// TIA Portal project "TCC" (V14)

(* hardware
DEVICE "S71500/ET200MP station_1"  S7-1500 station
   slot 0: "Rail_0"  Rack  6ES7 590-1***0-0AA0
   slot 1: "Selection"  CPU 1516-3 PN/DP  6ES7 516-3AN01-0AB0  V2.1
      slot 3: "CPU display_1"  6ES7591-1BA00-0AA0
   slot 2: "DI 32x24VDC HF_1"  DI 32x24VDC HF  6ES7 521-1BL00-0AB0  V2.1
   slot 3: "DQ 32x24VDC/0.5A HF_1"  DQ 32x24VDC/0.5A HF  6ES7 522-1BL01-0AB0  V1.0
   slot 4: "AI 8xU/I/RTD/TC ST_1"  AI 8xU/I/RTD/TC ST  6ES7 531-7KF00-0AB0  V2.1
   slot 5: "AQ 4xU/I ST_1"  AQ 4xU/I ST  6ES7 532-5HD00-0AB0  V2.1
DEVICE "S71500/ET200MP station_2"  S7-1500 station
   slot 0: "Rail_0"  Rack  6ES7 590-1***0-0AA0
   slot 1: "Handling-Assembly-Storage"  CPU 1516-3 PN/DP  6ES7 516-3AN01-0AB0  V2.1
      slot 3: "CPU display_1"  6ES7591-1BA00-0AA0
   slot 2: "DI 32x24VDC HF_1"  DI 32x24VDC HF  6ES7 521-1BL00-0AB0  V2.1
   slot 3: "DQ 32x24VDC/0.5A HF_1"  DQ 32x24VDC/0.5A HF  6ES7 522-1BL01-0AB0  V1.0
   slot 4: "AI 8xU/I/RTD/TC ST_1"  AI 8xU/I/RTD/TC ST  6ES7 531-7KF00-0AB0  V2.1
   slot 5: "AQ 4xU/I ST_1"  AQ 4xU/I ST  6ES7 532-5HD00-0AB0  V2.1
   slot 6: "TM Count 2x24V_1"  TM Count 2x24V  6ES7 550-1AA00-0AB0  V1.1
*)

// ===== PLC "Selection"  CPU 1516-3 PN/DP =====

VAR_GLOBAL   // PLC tag table "Default tag table"
   "Clock_Byte" AT %MB25 : Byte;
   "Clock_10Hz" AT %M25.0 : Bool;
   "Clock_5Hz" AT %M25.1 : Bool;
   "Clock_2.5Hz" AT %M25.2 : Bool;
   "Clock_2Hz" AT %M25.3 : Bool;
   "Clock_1.25Hz" AT %M25.4 : Bool;
   "Clock_1Hz" AT %M25.5 : Bool;
   "Clock_0.625Hz" AT %M25.6 : Bool;
   "Clock_0.5Hz" AT %M25.7 : Bool;
END_VAR

VAR_GLOBAL   // PLC tag table "IOTAGS"
   "I_MAG1EXT" AT %I0.0 : Bool;   // MAG 1 Cylinder Extended
   "I_MAG1RET" AT %I0.1 : Bool;   // MAG 1 Cylinder Retracted
   "I_MAG1EMPT" AT %I0.2 : Bool;   // MAG 1 Empty
   "I_MAG2EXT" AT %I0.3 : Bool;   // MAG 2 Cylinder Extended
   "I_MAG2RET" AT %I0.4 : Bool;   // MAG 2 Cylinder Retracted
   "I_MAG2EMPT" AT %I0.5 : Bool;   // MAG 2 Empty
   "I_PSLD" AT %I2.0 : Bool;   // Proximity Sensor Left Discharge Cylinder
   "I_PSCD" AT %I2.1 : Bool;   // Proximity Sensor Center Discharge Cylinder
   "I_PSRD" AT %I2.2 : Bool;   // Proximity Sensor Right Discharge Cylinder
   "I_RELAY1" AT %I2.3 : Bool;   // Relay
   "I_LDCEXT" AT %I1.0 : Bool;   // Left Discharge Cylinder Extended
   "I_LDCRET" AT %I1.1 : Bool;   // Left Discharge Cylinder Retracted
   "I_CDCEXT" AT %I1.2 : Bool;   // Center Discharge Cylinder Extended
   "I_CDCRET" AT %I1.3 : Bool;   // Center Discharge Cylinder Retracted
   "I_RDCEXT" AT %I1.4 : Bool;   // Right Discharge Cylinder Extended
   "I_RDCRET" AT %I1.5 : Bool;   // Right Discharge Cylinder Retracted
   "I_WHIT" AT %I1.6 : Bool;   // White Color Sensor
   "I_METAL" AT %I1.7 : Bool;   // Metalic Sensor
   "I_PSEOC" AT %I0.6 : Bool;   // Proximity Sensor End Of Conveyor Belt
   "I_DS" AT %IW4 : Word;   // Distance Sensor
   "O_MAG1EXT" AT %Q1.0 : Bool;   // Extend MAG 1 Cylinder
   "O_MAG1RET" AT %Q1.1 : Bool;   // Retract MAG 1 Cylinder
   "O_MAG2EXT" AT %Q1.2 : Bool;   // Extend MAG 2 Cylinder
   "O_MAG2RET" AT %Q1.3 : Bool;   // Retra MAG 2 Cylinder
   "O_RDCEXT" AT %Q0.2 : Bool;   // Extend Right Discharge Cylinder
   "O_CDCEXT" AT %Q0.1 : Bool;   // Extend Center Discharge Cylinder
   "O_LDCEXT" AT %Q0.0 : Bool;   // Extend Left Discharge Cylinder
   "O_CBFW" AT %Q1.4 : Bool;   // Conveyor Belt Forward
   "O_CBREV" AT %Q1.5 : Bool;   // Conveyor Belt Reverse
END_VAR

VAR_GLOBAL   // PLC tag table "Places"
   "p0" AT %M0.0 : Bool;
   "p1" AT %M0.1 : Bool;
   "p2" AT %M0.2 : Bool;
   "p3" AT %M0.3 : Bool;
   "p4" AT %M0.4 : Bool;
   "p5" AT %M0.5 : Bool;
   "p6" AT %M0.6 : Bool;
   "p7" AT %M0.7 : Bool;
   "p8" AT %M1.0 : Bool;
   "p9" AT %M1.1 : Bool;
   "p10" AT %M1.2 : Bool;
   "p11" AT %M1.3 : Bool;
   "p12" AT %M1.4 : Bool;
   "p27" AT %M1.6 : Bool;
   "p28" AT %M1.7 : Bool;
   "p29" AT %M2.0 : Bool;
   "p30" AT %M2.1 : Bool;
   "p31" AT %M2.2 : Bool;
   "p32" AT %M2.3 : Bool;
   "p33" AT %M2.4 : Bool;
   "p34" AT %M2.5 : Bool;
   "p35" AT %M2.6 : Bool;
   "p36" AT %M2.7 : Bool;
   "p37" AT %M3.0 : Bool;
   "p38" AT %M3.1 : Bool;
   "p39" AT %M3.2 : Bool;
   "p40" AT %M3.3 : Bool;
   "p41" AT %M3.4 : Bool;
   "p42" AT %M3.5 : Bool;
   "p43" AT %M3.6 : Bool;
   "p44" AT %M3.7 : Bool;
   "p45" AT %M4.0 : Bool;
   "p46" AT %M4.1 : Bool;
   "p47" AT %M4.2 : Bool;
   "p48" AT %M4.3 : Bool;
   "p49" AT %M4.4 : Bool;
   "p50" AT %M4.5 : Bool;
   "p51" AT %M4.6 : Bool;
   "p52" AT %M4.7 : Bool;
   "p53" AT %M5.0 : Bool;
   "p54" AT %M5.1 : Bool;
   "p55" AT %M5.2 : Bool;
   "p56" AT %M5.3 : Bool;
   "p57" AT %M5.4 : Bool;
   "p58" AT %M5.5 : Bool;
   "p59" AT %M5.6 : Bool;
   "p60" AT %M5.7 : Bool;
   "p61" AT %M6.0 : Bool;
   "p62" AT %M6.1 : Bool;
   "p63" AT %M6.2 : Bool;
   "p64" AT %M6.3 : Bool;
   "p65" AT %M6.4 : Bool;
   "p66" AT %M6.5 : Bool;
   "p67" AT %M6.6 : Bool;
   "p68" AT %M6.7 : Bool;
   "p69" AT %M7.0 : Bool;
   "p70" AT %M7.1 : Bool;
   "p71" AT %M7.2 : Bool;
   "p72" AT %M7.3 : Bool;
   "p73" AT %M7.4 : Bool;
END_VAR

VAR_GLOBAL   // PLC tag table "Transitions"
   "t0" AT %M7.5 : Bool;
   "t1" AT %M7.6 : Bool;
   "t2" AT %M7.7 : Bool;
   "t3" AT %M8.0 : Bool;
   "t4" AT %M8.1 : Bool;
   "t5" AT %M8.2 : Bool;
   "t6" AT %M8.3 : Bool;
   "t7" AT %M8.4 : Bool;
   "t18" AT %M8.5 : Bool;
   "t19" AT %M8.6 : Bool;
   "t20" AT %M8.7 : Bool;
   "t21" AT %M9.0 : Bool;
   "t22" AT %M9.1 : Bool;
   "t23" AT %M9.2 : Bool;
   "t24" AT %M9.3 : Bool;
   "t25" AT %M9.4 : Bool;
   "t26" AT %M9.5 : Bool;
   "t27" AT %M9.6 : Bool;
   "t28" AT %M9.7 : Bool;
   "t29" AT %M10.0 : Bool;
   "t30" AT %M10.1 : Bool;
   "t31" AT %M10.2 : Bool;
   "t32" AT %M10.3 : Bool;
   "t33" AT %M10.4 : Bool;
   "t34" AT %M10.5 : Bool;
   "t35" AT %M10.6 : Bool;
   "t36" AT %M10.7 : Bool;
   "t37" AT %M11.0 : Bool;
   "t38" AT %M11.1 : Bool;
   "t39" AT %M11.2 : Bool;
   "t40" AT %M11.3 : Bool;
   "t41" AT %M11.4 : Bool;
   "t42" AT %M11.5 : Bool;
   "t43" AT %M11.6 : Bool;
   "t44" AT %M11.7 : Bool;
   "t45" AT %M12.0 : Bool;
   "t46" AT %M12.1 : Bool;
   "t47" AT %M12.2 : Bool;
   "t48" AT %M12.3 : Bool;
   "t49" AT %M12.4 : Bool;
   "t50" AT %M12.5 : Bool;
   "t51" AT %M12.6 : Bool;
   "t52" AT %M12.7 : Bool;
   "t53" AT %M13.0 : Bool;
   "t54" AT %M13.1 : Bool;
   "t55" AT %M13.2 : Bool;
   "t56" AT %M13.3 : Bool;
   "t57" AT %M13.4 : Bool;
   "t58" AT %M13.5 : Bool;
   "t59" AT %M13.6 : Bool;
   "t60" AT %M13.7 : Bool;
   "t61" AT %M14.0 : Bool;
   "t62" AT %M14.1 : Bool;
   "t63" AT %M14.2 : Bool;
   "t64" AT %M14.3 : Bool;
   "t65" AT %M14.4 : Bool;
   "t66" AT %M14.5 : Bool;
   "t67" AT %M14.6 : Bool;
   "t68" AT %M14.7 : Bool;
   "t69" AT %M15.0 : Bool;
   "t70" AT %M15.1 : Bool;
   "t71" AT %M15.2 : Bool;
END_VAR

VAR_GLOBAL   // PLC tag table "Auxiliar"
   "PresenceR" AT %M15.3 : Bool;
   "ConcUP" AT %M15.4 : Bool;
   "ConcDWN" AT %M15.5 : Bool;
   "Presence_prev" AT %M15.6 : Bool;
   "I_PSEOCr_prev" AT %M15.7 : Bool;
   "PSEOCR" AT %M16.0 : Bool;
   "PSEOCF" AT %M16.1 : Bool;
   "BTInit" AT %M24.0 : Bool;
   "BTStart" AT %M24.1 : Bool;
   "BTSTOP" AT %M24.2 : Bool;
   "btget" AT %M24.3 : Bool;
   "bini" AT %M1.5 : Bool;
   "clkprev" AT %M24.4 : Bool;
   "I_PSEOCf_prev" AT %M24.6 : Bool;
END_VAR

VAR_GLOBAL   // PLC tag table "Conditions"
   "b0" AT %M16.2 : Bool;
   "b1" AT %M16.3 : Bool;
   "b2" AT %M16.4 : Bool;
   "b3" AT %M16.5 : Bool;
   "b4" AT %M16.6 : Bool;
   "b5" AT %M16.7 : Bool;
   "b6" AT %M17.0 : Bool;
   "b7" AT %M17.1 : Bool;
   "b18" AT %M17.2 : Bool;
   "b19" AT %M17.3 : Bool;
   "b20" AT %M17.4 : Bool;
   "b21" AT %M17.5 : Bool;
   "b22" AT %M17.6 : Bool;
   "b23" AT %M17.7 : Bool;
   "b24" AT %M18.0 : Bool;
   "b25" AT %M18.1 : Bool;
   "b26" AT %M18.2 : Bool;
   "b27" AT %M18.3 : Bool;
   "b28" AT %M18.4 : Bool;
   "b29" AT %M18.5 : Bool;
   "b30" AT %M18.6 : Bool;
   "b31" AT %M18.7 : Bool;
   "b32" AT %M19.0 : Bool;
   "b33" AT %M19.1 : Bool;
   "b34" AT %M19.2 : Bool;
   "b35" AT %M19.3 : Bool;
   "b36" AT %M19.4 : Bool;
   "b37" AT %M19.5 : Bool;
   "b38" AT %M19.6 : Bool;
   "b39" AT %M19.7 : Bool;
   "b40" AT %M20.0 : Bool;
   "b41" AT %M20.1 : Bool;
   "b42" AT %M20.2 : Bool;
   "b43" AT %M20.3 : Bool;
   "b44" AT %M20.4 : Bool;
   "b45" AT %M20.5 : Bool;
   "b46" AT %M20.6 : Bool;
   "b47" AT %M20.7 : Bool;
   "b48" AT %M21.0 : Bool;
   "b49" AT %M21.1 : Bool;
   "b50" AT %M21.2 : Bool;
   "b51" AT %M21.3 : Bool;
   "b52" AT %M21.4 : Bool;
   "b53" AT %M21.5 : Bool;
   "b54" AT %M21.6 : Bool;
   "b55" AT %M21.7 : Bool;
   "b56" AT %M22.0 : Bool;
   "b57" AT %M22.1 : Bool;
   "b58" AT %M22.2 : Bool;
   "b59" AT %M22.3 : Bool;
   "b60" AT %M22.4 : Bool;
   "b61" AT %M22.5 : Bool;
   "b62" AT %M22.6 : Bool;
   "b63" AT %M22.7 : Bool;
   "b64" AT %M23.0 : Bool;
   "b65" AT %M23.1 : Bool;
   "b66" AT %M23.2 : Bool;
   "b67" AT %M23.3 : Bool;
   "b68" AT %M23.4 : Bool;
   "b69" AT %M23.5 : Bool;
   "b70" AT %M23.6 : Bool;
   "b71" AT %M23.7 : Bool;
   "b162" AT %M24.5 : Bool;
   "b156_StopAll" AT %M24.7 : Bool;
END_VAR

VAR_GLOBAL   // PLC tag table "Logging"
   "AcqRun" AT %M26.0 : Bool;
   "stopAcquisition" AT %M26.2 : Bool;
   "DataLogCreated" AT %M26.3 : Bool;
   "Done_Signal" AT %M26.4 : Bool;
   "Busy" AT %M26.5 : Bool;
   "Error" AT %M26.6 : Bool;
   "Status" AT %MW28 : Word;
   "LogTimeElapsed" AT %MD30 : Time;
   "AcqNewValues" AT %M26.7 : Bool;
   "Done_Open" AT %M27.0 : Bool;
   "Busy_Open" AT %M27.1 : Bool;
   "Error_Open" AT %M27.2 : Bool;
   "Status_Open" AT %MW34 : Word;
   "Done_Write" AT %M36.0 : Bool;
   "Busy_Write" AT %M36.1 : Bool;
   "Error_Write" AT %M36.2 : Bool;
   "Status_Write" AT %MW38 : Word;
   "closeDL" AT %M27.3 : Bool;
   "startAcquisition" AT %M26.1 : Bool;
   "DeleteDl" AT %M27.4 : Bool;
   "startAcqprev" AT %M27.5 : Bool;
END_VAR

// folder: Logging

DATA_BLOCK "LOGDATA_DB"   // DB18
{ S7_Optimized_Access := 'TRUE' }
VERSION : 0.1
// stored: InstanceOfName LOGDATA
"LOGDATA"
BEGIN
END_DATA_BLOCK

DATA_BLOCK "IOVEC_FROMPLC2"   // DB19
{ S7_Optimized_Access := 'FALSE' }
VERSION : 0.1
   VAR
      I_SDO : Bool;
      I_SDC : Bool;
      I_AUHEXT : Bool;
      I_AUHRET : Bool;
      I_INDARM : Bool;
      I_ARMLOW : Bool;
      I_ARMHIG : Bool;
      I_ARMRET : Bool;
      I_ARMEXT : Bool;
      I_SUVE : Bool;
      I_SUILS : Bool;
      I_SUSLS : Bool;
      I_SUEXT : Bool;
      I_SURET : Bool;
      I_RELAY2 : Bool;
      I_SUHE : Bool;
      I_SURLS : Bool;
      I_SULLS : Bool;
      I_SUARMALE : Bool;
      O_SDO : Bool;
      O_SDC : Bool;
      O_AUHRET : Bool;
      O_AUHEXT : Bool;
      O_PRESSLOW : Bool;
      O_PRESSHIG : Bool;
      O_ARMHIG : Bool;
      O_VACON : Bool;
      O_ARMEXT : Bool;
      O_ARMCCW : Bool;
      O_ARMCW : Bool;
      O_SUEXT : Bool;
      O_SUUP : Bool;
      O_SUDWN : Bool;
      O_SURIGHT : Bool;
      O_SULEFT : Bool;
   END_VAR
BEGIN
END_DATA_BLOCK

DATA_BLOCK "DATALOGDATA"   // DB21
{ S7_Optimized_Access := 'TRUE' }
VERSION : 0.1
   VAR
      IOVECNAMES : Array[0..64] of String;
      IOVEC : Array[0..64] of Bool;
      AcqValues : Array[0..64] of Bool;
      AcqValuesprev : Array[0..64] of Bool;
      Data : Struct
         I_MAG1EXT : Bool;
         I_MAG1RET : Bool;
         I_MAG1EMPT : Bool;
         I_MAG2EXT : Bool;
         I_MAG2RET : Bool;
         I_MAG2EMPT : Bool;
         I_PSLD : Bool;
         I_PSCD : Bool;
         I_PSRD : Bool;
         I_RELAY1 : Bool;
         I_LDCEXT : Bool;
         I_LDCRET : Bool;
         I_CDCEXT : Bool;
         I_CDCRET : Bool;
         I_RDCEXT : Bool;
         I_RDCRET : Bool;
         I_WHIT : Bool;
         I_METAL : Bool;
         I_PSEOC : Bool;
         ConcDWN : Bool;
         ConcUP : Bool;
         O_MAG1EXT : Bool;
         O_MAG1RET : Bool;
         O_MAG2EXT : Bool;
         O_MAG2RET : Bool;
         O_RDCEXT : Bool;
         O_CDCEXT : Bool;
         O_LDCEXT : Bool;
         O_CBFW : Bool;
         O_CBREV : Bool;
         I_SDO : Bool;
         I_SDC : Bool;
         I_AUHEXT : Bool;
         I_AUHRET : Bool;
         I_INDARM : Bool;
         I_ARMLOW : Bool;
         I_ARMHIG : Bool;
         I_ARMRET : Bool;
         I_ARMEXT : Bool;
         I_SUVE : Bool;
         I_SUILS : Bool;
         I_SUSLS : Bool;
         I_SUEXT : Bool;
         I_SURET : Bool;
         I_RELAY2 : Bool;
         I_SUHE : Bool;
         I_SURLS : Bool;
         I_SULLS : Bool;
         I_SUARMALE : Bool;
         O_SDO : Bool;
         O_SDC : Bool;
         O_AUHRET : Bool;
         O_AUHEXT : Bool;
         O_PRESSLOW : Bool;
         O_PRESSHIG : Bool;
         O_ARMHIG : Bool;
         O_VACON : Bool;
         O_ARMEXT : Bool;
         O_ARMCCW : Bool;
         O_ARMCW : Bool;
         O_SUEXT : Bool;
         O_SUUP : Bool;
         O_SUDWN : Bool;
         O_SURIGHT : Bool;
         O_SULEFT : Bool;
      END_STRUCT;
      header : String;
      ID : DWord;
      "Name" : String;
   END_VAR
BEGIN
   IOVECNAMES[1] := '1';
   IOVECNAMES[2] := '2';
   IOVECNAMES[3] := '3';
   IOVECNAMES[4] := '4';
   IOVECNAMES[5] := '5';
   IOVECNAMES[6] := '6';
   IOVECNAMES[7] := '7';
   IOVECNAMES[8] := '8';
   IOVECNAMES[9] := '9';
   IOVECNAMES[10] := '10';
   IOVECNAMES[11] := '11';
   IOVECNAMES[12] := '12';
   IOVECNAMES[13] := '13';
   IOVECNAMES[14] := '14';
   IOVECNAMES[15] := '15';
   IOVECNAMES[16] := '16';
   IOVECNAMES[17] := '17';
   IOVECNAMES[18] := '18';
   IOVECNAMES[19] := '19';
   IOVECNAMES[20] := '20';
   IOVECNAMES[21] := '21';
   IOVECNAMES[22] := '22';
   IOVECNAMES[0] := '0';
   IOVECNAMES[23] := '23';
   IOVECNAMES[24] := '24';
   IOVECNAMES[25] := '25';
   IOVECNAMES[26] := '26';
   IOVECNAMES[27] := '27';
   IOVECNAMES[28] := '28';
   IOVECNAMES[29] := '29';
   IOVECNAMES[30] := '30';
   IOVECNAMES[31] := '31';
   IOVECNAMES[32] := '32';
   IOVECNAMES[33] := '33';
   IOVECNAMES[34] := '34';
   IOVECNAMES[35] := '35';
   IOVECNAMES[36] := '36';
   IOVECNAMES[37] := '37';
   IOVECNAMES[38] := '38';
   IOVECNAMES[39] := '39';
   IOVECNAMES[40] := '40';
   IOVECNAMES[41] := '41';
   IOVECNAMES[42] := '42';
   IOVECNAMES[43] := '43';
   IOVECNAMES[44] := '44';
   IOVECNAMES[45] := '45';
   IOVECNAMES[46] := '46';
   IOVECNAMES[47] := '47';
   IOVECNAMES[48] := '48';
   IOVECNAMES[49] := '49';
   IOVECNAMES[50] := '50';
   IOVECNAMES[51] := '51';
   IOVECNAMES[52] := '52';
   IOVECNAMES[53] := '53';
   IOVECNAMES[54] := '54';
   IOVECNAMES[55] := '55';
   IOVECNAMES[56] := '56';
   IOVECNAMES[57] := '57';
   IOVECNAMES[58] := '58';
   IOVECNAMES[59] := '59';
   IOVECNAMES[60] := '60';
   IOVECNAMES[61] := '61';
   IOVECNAMES[62] := '62';
   IOVECNAMES[63] := '63';
   IOVECNAMES[64] := '64';
END_DATA_BLOCK

// folder: PetriNet

DATA_BLOCK "FROM_PLC2"   // DB4
{ S7_Optimized_Access := 'FALSE' }
VERSION : 0.1
   VAR
      p13 : Bool;
      p17 : Bool;
      p26 : Bool;
      p14 : Bool;
      p18 : Bool;
      p107 : Bool;
      p0 : Bool;
      b162aux : Bool;
   END_VAR
BEGIN
END_DATA_BLOCK

DATA_BLOCK "TO_PLC2"   // DB5
{ S7_Optimized_Access := 'FALSE' }
VERSION : 0.1
   VAR
      b0 : Bool;
      b18 : Bool;
      b19 : Bool;
      b71 : Bool;
      b45 : Bool;
      b162 : Bool;
      btStopOn : Bool;
      btStopOff : Bool;
   END_VAR
BEGIN
END_DATA_BLOCK

// folder: PetriNet/TimedTransitions

DATA_BLOCK "t7_time"   // DB1
{ S7_Optimized_Access := 'TRUE' }
AUTHOR : Simatic
FAMILY : IEC
NAME : IEC_TMR
VERSION : 1.0
// stored: InstanceOfName IEC_TIMER
"IEC_TIMER"
BEGIN
END_DATA_BLOCK

DATA_BLOCK "t24_time"   // DB6
{ S7_Optimized_Access := 'TRUE' }
AUTHOR : Simatic
FAMILY : IEC
NAME : IEC_TMR
VERSION : 1.0
// stored: InstanceOfName IEC_TIMER
"IEC_TIMER"
BEGIN
END_DATA_BLOCK

DATA_BLOCK "t25_time"   // DB7
{ S7_Optimized_Access := 'TRUE' }
AUTHOR : Simatic
FAMILY : IEC
NAME : IEC_TMR
VERSION : 1.0
// stored: InstanceOfName IEC_TIMER
"IEC_TIMER"
BEGIN
END_DATA_BLOCK

DATA_BLOCK "t43_time"   // DB8
{ S7_Optimized_Access := 'TRUE' }
AUTHOR : Simatic
FAMILY : IEC
NAME : IEC_TMR
VERSION : 1.0
// stored: InstanceOfName IEC_TIMER
"IEC_TIMER"
BEGIN
END_DATA_BLOCK

DATA_BLOCK "t50_time"   // DB9
{ S7_Optimized_Access := 'TRUE' }
AUTHOR : Simatic
FAMILY : IEC
NAME : IEC_TMR
VERSION : 1.0
// stored: InstanceOfName IEC_TIMER
"IEC_TIMER"
BEGIN
END_DATA_BLOCK

DATA_BLOCK "t51_time"   // DB10
{ S7_Optimized_Access := 'TRUE' }
AUTHOR : Simatic
FAMILY : IEC
NAME : IEC_TMR
VERSION : 1.0
// stored: InstanceOfName IEC_TIMER
"IEC_TIMER"
BEGIN
END_DATA_BLOCK

DATA_BLOCK "t69_time"   // DB11
{ S7_Optimized_Access := 'TRUE' }
AUTHOR : Simatic
FAMILY : IEC
NAME : IEC_TMR
VERSION : 1.0
// stored: InstanceOfName IEC_TIMER
"IEC_TIMER"
BEGIN
END_DATA_BLOCK

// folder: System blocks/Program resources

DATA_BLOCK "LogTime"   // DB12
{ S7_Optimized_Access := 'TRUE' }
AUTHOR : Simatic
FAMILY : IEC
NAME : IEC_TMR
VERSION : 1.0
// stored: InstanceOfName IEC_TIMER
"IEC_TIMER"
BEGIN
END_DATA_BLOCK

// folder: (top level)

ORGANIZATION_BLOCK "Main"   // OB1, LAD, ProgramCycle
TITLE = "Main Program Sweep (Cycle)"
{ S7_Optimized_Access := 'TRUE' }
VERSION : 0.1
   VAR_INPUT
      Initial_Call : Bool;   // Initial call of this OB
      Remanence : Bool;   // =True, if remanent data are available
   END_VAR
BEGIN

REGION Network 1: GET VALUES FROM OTHER PLC
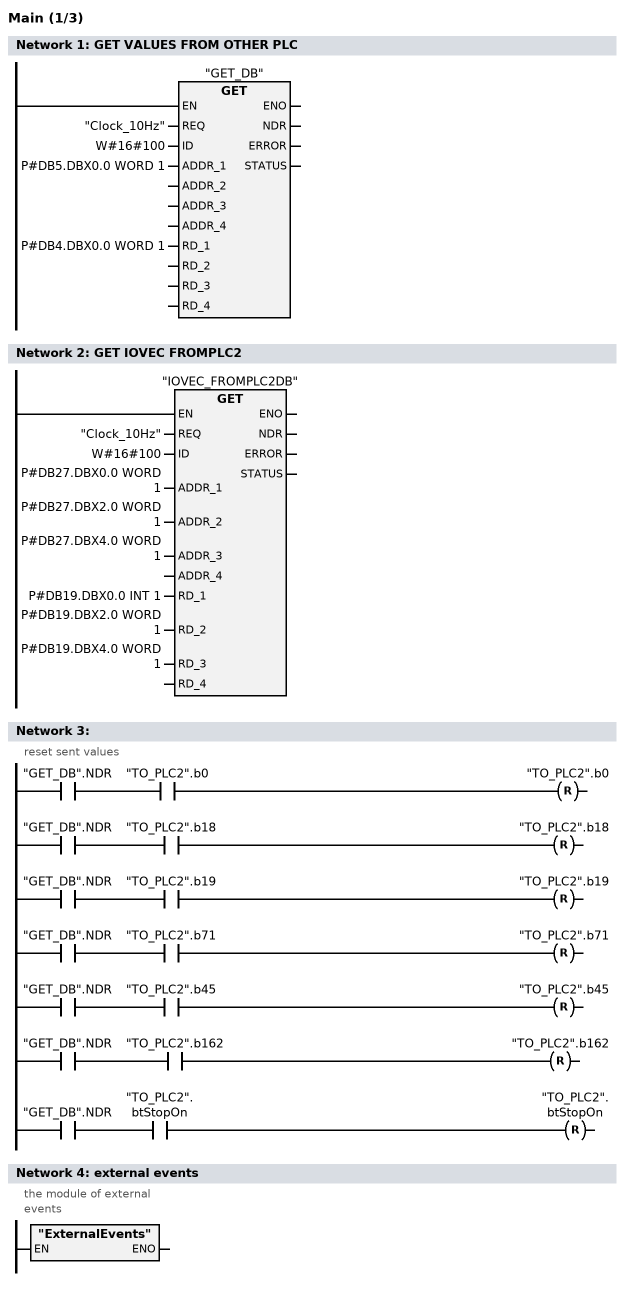
   "GET_DB"(REQ := "Clock_10Hz", ID := W#16#100, ADDR_1 := P#DB5.DBX0.0 WORD 1, RD_1 := P#DB4.DBX0.0 WORD 1);   // GET
END_REGION

REGION Network 2: GET IOVEC FROMPLC2
   "IOVEC_FROMPLC2DB"(REQ := "Clock_10Hz",   // GET
                      ID := W#16#100,
                      ADDR_1 := P#DB27.DBX0.0 WORD 1,
                      ADDR_2 := P#DB27.DBX2.0 WORD 1,
                      ADDR_3 := P#DB27.DBX4.0 WORD 1,
                      RD_1 := P#DB19.DBX0.0 INT 1,
                      RD_2 := P#DB19.DBX2.0 WORD 1,
                      RD_3 := P#DB19.DBX4.0 WORD 1);
END_REGION

REGION Network 3
   // reset sent values
   RUNG wire#powerrail
      Contact( "GET_DB".NDR )
      Contact( "TO_PLC2".b0 )
      R_Coil( "TO_PLC2".b0 )
   END_RUNG
   RUNG wire#powerrail
      Contact( "GET_DB".NDR )
      Contact( "TO_PLC2".b18 )
      R_Coil( "TO_PLC2".b18 )
   END_RUNG
   RUNG wire#powerrail
      Contact( "GET_DB".NDR )
      Contact( "TO_PLC2".b19 )
      R_Coil( "TO_PLC2".b19 )
   END_RUNG
   RUNG wire#powerrail
      Contact( "GET_DB".NDR )
      Contact( "TO_PLC2".b71 )
      R_Coil( "TO_PLC2".b71 )
   END_RUNG
   RUNG wire#powerrail
      Contact( "GET_DB".NDR )
      Contact( "TO_PLC2".b45 )
      R_Coil( "TO_PLC2".b45 )
   END_RUNG
   RUNG wire#powerrail
      Contact( "GET_DB".NDR )
      Contact( "TO_PLC2".b162 )
      R_Coil( "TO_PLC2".b162 )
   END_RUNG
   RUNG wire#powerrail
      Contact( "GET_DB".NDR )
      Contact( "TO_PLC2".btStopOn )
      R_Coil( "TO_PLC2".btStopOn )
   END_RUNG
   // the same network as SCL:
   IF "GET_DB".NDR AND "TO_PLC2".b0 THEN "TO_PLC2".b0 := FALSE; END_IF;
   IF "GET_DB".NDR AND "TO_PLC2".b18 THEN "TO_PLC2".b18 := FALSE; END_IF;
   IF "GET_DB".NDR AND "TO_PLC2".b19 THEN "TO_PLC2".b19 := FALSE; END_IF;
   IF "GET_DB".NDR AND "TO_PLC2".b71 THEN "TO_PLC2".b71 := FALSE; END_IF;
   IF "GET_DB".NDR AND "TO_PLC2".b45 THEN "TO_PLC2".b45 := FALSE; END_IF;
   IF "GET_DB".NDR AND "TO_PLC2".b162 THEN "TO_PLC2".b162 := FALSE; END_IF;
   IF "GET_DB".NDR AND "TO_PLC2".btStopOn THEN "TO_PLC2".btStopOn := FALSE; END_IF;
END_REGION

REGION Network 4: external events
   // the module of external
   // events
   RUNG wire#powerrail
      "ExternalEvents"()
   END_RUNG
   // the same network as SCL:
   "ExternalEvents"();
END_REGION

REGION Network 5: conditions
   // the module of firing conditions
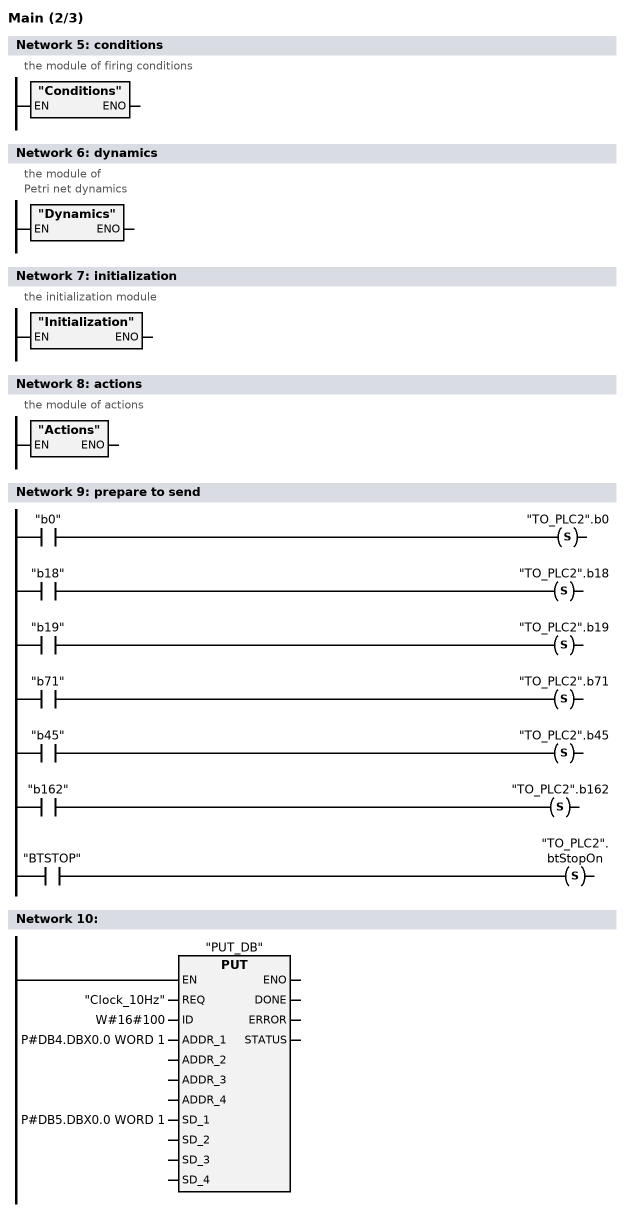
   RUNG wire#powerrail
      "Conditions"()
   END_RUNG
   // the same network as SCL:
   "Conditions"();
END_REGION

REGION Network 6: dynamics
   // the module of
   // Petri net dynamics
   RUNG wire#powerrail
      "Dynamics"()
   END_RUNG
   // the same network as SCL:
   "Dynamics"();
END_REGION

REGION Network 7: initialization
   // the initialization module
   RUNG wire#powerrail
      "Initialization"()
   END_RUNG
   // the same network as SCL:
   "Initialization"();
END_REGION

REGION Network 8: actions
   // the module of actions
   RUNG wire#powerrail
      "Actions"()
   END_RUNG
   // the same network as SCL:
   "Actions"();
END_REGION

REGION Network 9: prepare to send
   RUNG wire#powerrail
      Contact( "b0" )
      S_Coil( "TO_PLC2".b0 )
   END_RUNG
   RUNG wire#powerrail
      Contact( "b18" )
      S_Coil( "TO_PLC2".b18 )
   END_RUNG
   RUNG wire#powerrail
      Contact( "b19" )
      S_Coil( "TO_PLC2".b19 )
   END_RUNG
   RUNG wire#powerrail
      Contact( "b71" )
      S_Coil( "TO_PLC2".b71 )
   END_RUNG
   RUNG wire#powerrail
      Contact( "b45" )
      S_Coil( "TO_PLC2".b45 )
   END_RUNG
   RUNG wire#powerrail
      Contact( "b162" )
      S_Coil( "TO_PLC2".b162 )
   END_RUNG
   RUNG wire#powerrail
      Contact( "BTSTOP" )
      S_Coil( "TO_PLC2".btStopOn )
   END_RUNG
   // the same network as SCL:
   IF "b0" THEN "TO_PLC2".b0 := TRUE; END_IF;
   IF "b18" THEN "TO_PLC2".b18 := TRUE; END_IF;
   IF "b19" THEN "TO_PLC2".b19 := TRUE; END_IF;
   IF "b71" THEN "TO_PLC2".b71 := TRUE; END_IF;
   IF "b45" THEN "TO_PLC2".b45 := TRUE; END_IF;
   IF "b162" THEN "TO_PLC2".b162 := TRUE; END_IF;
   IF "BTSTOP" THEN "TO_PLC2".btStopOn := TRUE; END_IF;
END_REGION

REGION Network 10
   "PUT_DB"(REQ := "Clock_10Hz", ID := W#16#100, ADDR_1 := P#DB4.DBX0.0 WORD 1, SD_1 := P#DB5.DBX0.0 WORD 1);   // PUT
END_REGION

REGION Network 11: LOG DATA
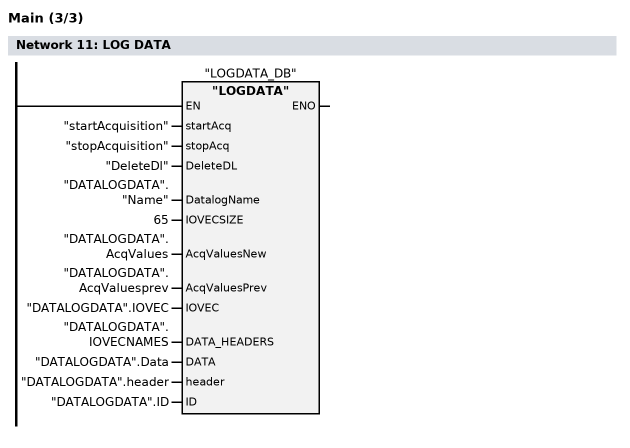
   RUNG wire#powerrail
      "LOGDATA_DB"(startAcq := "startAcquisition", stopAcq := "stopAcquisition", DeleteDL := "DeleteDl", DatalogName := "DATALOGDATA"."Name", IOVECSIZE := 65, AcqValuesNew := "DATALOGDATA".AcqValues, AcqValuesPrev := "DATALOGDATA".AcqValuesprev, IOVEC := "DATALOGDATA".IOVEC, DATA_HEADERS := "DATALOGDATA".IOVECNAMES, DATA := "DATALOGDATA".Data, header := "DATALOGDATA".header, ID := "DATALOGDATA".ID)
   END_RUNG
   // the same network as SCL:
   "LOGDATA_DB"(startAcq := "startAcquisition",   // "LOGDATA"
                stopAcq := "stopAcquisition",
                DeleteDL := "DeleteDl",
                DatalogName := "DATALOGDATA"."Name",
                IOVECSIZE := 65,
                AcqValuesNew := "DATALOGDATA".AcqValues,
                AcqValuesPrev := "DATALOGDATA".AcqValuesprev,
                IOVEC := "DATALOGDATA".IOVEC,
                DATA_HEADERS := "DATALOGDATA".IOVECNAMES,
                DATA := "DATALOGDATA".Data,
                header := "DATALOGDATA".header,
                ID := "DATALOGDATA".ID);
END_REGION
END_ORGANIZATION_BLOCK

// folder: Logging

FUNCTION_BLOCK "LOGDATA"   // FB1, LAD
{ S7_Optimized_Access := 'TRUE' }
VERSION : 0.1
   VAR_INPUT
      startAcq : Bool;
      stopAcq : Bool;
      DeleteDL : Bool;
      DatalogName : String;
      IOVECSIZE : UDInt;
   END_VAR
   VAR_IN_OUT
      AcqValuesNew : Array[*] of Bool;
      AcqValuesPrev : Array[*] of Bool;
      IOVEC : Array[*] of Bool;
      DATA_HEADERS : Array[*] of String;
      DATA : Variant;
      header : String;
      ID : DWord;
   END_VAR
   VAR_TEMP
      DeleteDatalog : Bool;
      moveBlkVariantRetVal : Int;
      i : Int;
      dataheaderslowerbound : DInt;
      dataheadersupperbound : DInt;
   END_VAR
   VAR_TEMP   // added for the SCL form of the ladder/FBD networks
      _w1 : Bool;
      _w2 : Bool;
   END_VAR
BEGIN

REGION Network 1 (SCL): Name header
       #header := '';
   #dataheaderslowerbound := LOWER_BOUND(ARR := #DATA_HEADERS, DIM := 1);
   #dataheadersupperbound := UPPER_BOUND(ARR := #DATA_HEADERS, DIM := 1);

   FOR #i := #dataheaderslowerbound TO #dataheadersupperbound-1 DO
       // Statement section FOR

       #header := CONCAT(IN1 := #header, IN2 := #DATA_HEADERS[#i]);
       #header := CONCAT(IN1 := #header, IN2 := ',');
   END_FOR;
   #header := CONCAT(IN1 := #header, IN2 := #DATA_HEADERS[#dataheadersupperbound]);
END_REGION

REGION Network 2: Start or stop acquisition
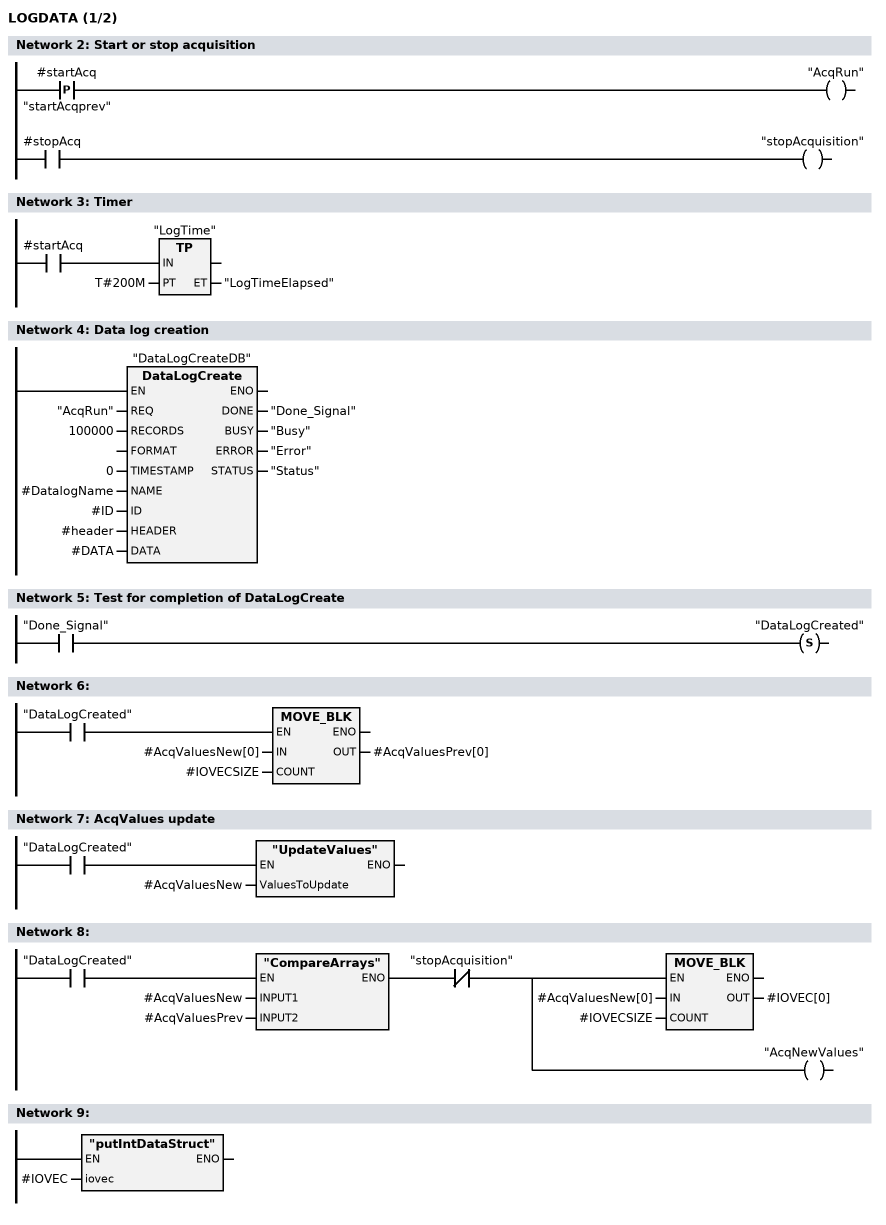
   RUNG wire#powerrail
      P_Contact(operand := #startAcq, bit := "startAcqprev")
      Coil( "AcqRun" )
   END_RUNG
   RUNG wire#powerrail
      Contact( #stopAcq )
      Coil( "stopAcquisition" )
   END_RUNG
   // the same network as SCL:
   #_w1 := #startAcq AND NOT "startAcqprev";   // rising edge of #startAcq
   "startAcqprev" := #startAcq;
   "AcqRun" := #_w1;
   "stopAcquisition" := #stopAcq;
END_REGION

REGION Network 3: Timer
   "LogTime".TP(IN := #startAcq, PT := T#200M, ET => "LogTimeElapsed");
END_REGION

REGION Network 4: Data log creation
   "DataLogCreateDB"(REQ := "AcqRun",   // DataLogCreate
                     RECORDS := 100000,
                     TIMESTAMP := 0,
                     "NAME" := #DatalogName,
                     ID := #ID,
                     HEADER := #header,
                     DATA := #DATA,
                     DONE => "Done_Signal",
                     BUSY => "Busy",
                     ERROR => "Error",
                     STATUS => "Status");
END_REGION

REGION Network 5: Test for completion of DataLogCreate
   RUNG wire#powerrail
      Contact( "Done_Signal" )
      S_Coil( "DataLogCreated" )
   END_RUNG
   // the same network as SCL:
   IF "Done_Signal" THEN "DataLogCreated" := TRUE; END_IF;
END_REGION

REGION Network 6
   IF "DataLogCreated" THEN
       MOVE_BLK(IN := #AcqValuesNew[0], COUNT := #IOVECSIZE, OUT => #AcqValuesPrev[0]);
   END_IF;
END_REGION

REGION Network 7: AcqValues update
   RUNG wire#powerrail
      Contact( "DataLogCreated" )
      "UpdateValues"(ValuesToUpdate := #AcqValuesNew)
   END_RUNG
   // the same network as SCL:
   IF "DataLogCreated" THEN "UpdateValues"(ValuesToUpdate := #AcqValuesNew); END_IF;
END_REGION

REGION Network 8
   "CompareArrays"(EN := "DataLogCreated", INPUT1 := #AcqValuesNew, INPUT2 := #AcqValuesPrev, ENO => #_w1);
   #_w2 := #_w1 AND NOT "stopAcquisition";
   IF #_w2 THEN MOVE_BLK(IN := #AcqValuesNew[0], COUNT := #IOVECSIZE, OUT => #IOVEC[0]); END_IF;
   "AcqNewValues" := #_w2;
END_REGION

REGION Network 9
   RUNG wire#powerrail
      "putIntDataStruct"(iovec := #IOVEC)
   END_RUNG
   // the same network as SCL:
   "putIntDataStruct"(iovec := #IOVEC);
END_REGION

REGION Network 10: Write to data log
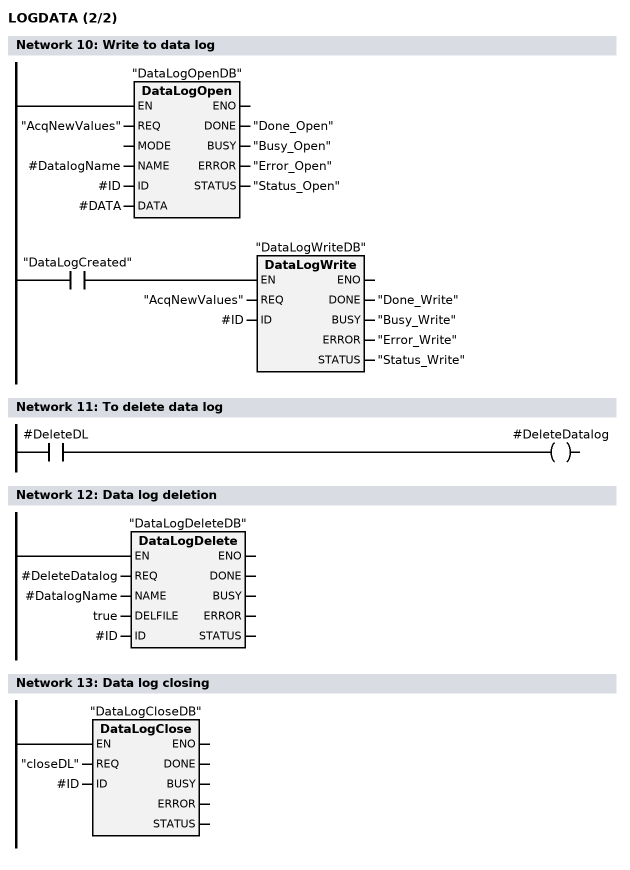
   "DataLogOpenDB"(REQ := "AcqNewValues",   // DataLogOpen
                   "NAME" := #DatalogName,
                   ID := #ID,
                   Data := #DATA,
                   DONE => "Done_Open",
                   BUSY => "Busy_Open",
                   ERROR => "Error_Open",
                   STATUS => "Status_Open");
   IF "DataLogCreated" THEN
       "DataLogWriteDB"(REQ := "AcqNewValues",   // DataLogWrite
                        ID := #ID,
                        DONE => "Done_Write",
                        BUSY => "Busy_Write",
                        ERROR => "Error_Write",
                        STATUS => "Status_Write");
   END_IF;
END_REGION

REGION Network 11: To delete data log
   RUNG wire#powerrail
      Contact( #DeleteDL )
      Coil( #DeleteDatalog )
   END_RUNG
   // the same network as SCL:
   #DeleteDatalog := #DeleteDL;
END_REGION

REGION Network 12: Data log deletion
   "DataLogDeleteDB"(REQ := #DeleteDatalog, "NAME" := #DatalogName, DelFile := true, ID := #ID);   // DataLogDelete
END_REGION

REGION Network 13: Data log closing
   "DataLogCloseDB"(REQ := "closeDL", ID := #ID);   // DataLogClose
END_REGION
END_FUNCTION_BLOCK

FUNCTION "UpdateValues" : Void   // FC6, LAD
{ S7_Optimized_Access := 'TRUE' }
VERSION : 0.1
   VAR_IN_OUT
      ValuesToUpdate : Array[*] of Bool;
   END_VAR
BEGIN

REGION Network 1 (SCL)
   #ValuesToUpdate[0] := "I_MAG1EXT";
   #ValuesToUpdate[1] := "I_MAG1RET";
   #ValuesToUpdate[2] := "I_MAG1EMPT";
   #ValuesToUpdate[3] := "I_MAG2EXT";
   #ValuesToUpdate[4] := "I_MAG2RET";
   #ValuesToUpdate[5] := "I_MAG2EMPT";
   #ValuesToUpdate[6] := "I_PSLD";
   #ValuesToUpdate[7] := "I_PSCD";
   #ValuesToUpdate[8] := "I_PSRD";
   #ValuesToUpdate[9] := "I_RELAY1";
   #ValuesToUpdate[10] := "I_LDCEXT";
   #ValuesToUpdate[11] := "I_LDCRET";
   #ValuesToUpdate[12] := "I_CDCEXT";
   #ValuesToUpdate[13] := "I_CDCRET";
   #ValuesToUpdate[14] := "I_RDCEXT";
   #ValuesToUpdate[15] := "I_RDCRET";
   #ValuesToUpdate[16] := "I_WHIT";
   #ValuesToUpdate[17] := "I_METAL";
   #ValuesToUpdate[18] := "I_PSEOC";
   #ValuesToUpdate[19] := "ConcDWN";
   #ValuesToUpdate[20] := "ConcUP";
   #ValuesToUpdate[21] := "O_MAG1EXT";
   #ValuesToUpdate[22] := "O_MAG1RET";
   #ValuesToUpdate[23] := "O_MAG2EXT";
   #ValuesToUpdate[24] := "O_MAG2RET";
   #ValuesToUpdate[25] := "O_RDCEXT";
   #ValuesToUpdate[26] := "O_CDCEXT";
   #ValuesToUpdate[27] := "O_LDCEXT";
   #ValuesToUpdate[28] := "O_CBFW";
   #ValuesToUpdate[29] := "O_CBREV";
   #ValuesToUpdate[30] := "IOVEC_FROMPLC2".I_SDO;
   #ValuesToUpdate[31] := "IOVEC_FROMPLC2".I_SDC;
   #ValuesToUpdate[32] := "IOVEC_FROMPLC2".I_AUHEXT;
   #ValuesToUpdate[33] := "IOVEC_FROMPLC2".I_AUHRET;
   #ValuesToUpdate[34] := "IOVEC_FROMPLC2".I_INDARM;
   #ValuesToUpdate[35] := "IOVEC_FROMPLC2".I_ARMLOW;
   #ValuesToUpdate[36] := "IOVEC_FROMPLC2".I_ARMHIG;
   #ValuesToUpdate[37] := "IOVEC_FROMPLC2".I_ARMRET;
   #ValuesToUpdate[38] := "IOVEC_FROMPLC2".I_ARMEXT;
   #ValuesToUpdate[39] := "IOVEC_FROMPLC2".I_SUVE;
   #ValuesToUpdate[40] := "IOVEC_FROMPLC2".I_SUILS;
   #ValuesToUpdate[41] := "IOVEC_FROMPLC2".I_SUSLS;
   #ValuesToUpdate[42] := "IOVEC_FROMPLC2".I_SUEXT;
   #ValuesToUpdate[43] := "IOVEC_FROMPLC2".I_SURET;
   #ValuesToUpdate[44] := "IOVEC_FROMPLC2".I_RELAY2;
   #ValuesToUpdate[45] := "IOVEC_FROMPLC2".I_SUHE;
   #ValuesToUpdate[46] := "IOVEC_FROMPLC2".I_SURLS;
   #ValuesToUpdate[47] := "IOVEC_FROMPLC2".I_SULLS;
   #ValuesToUpdate[48] := "IOVEC_FROMPLC2".I_SUARMALE;
   #ValuesToUpdate[49] := "IOVEC_FROMPLC2".O_SDO;
   #ValuesToUpdate[50] := "IOVEC_FROMPLC2".O_SDC;
   #ValuesToUpdate[51] := "IOVEC_FROMPLC2".O_AUHRET;
   #ValuesToUpdate[52] := "IOVEC_FROMPLC2".O_AUHEXT;
   #ValuesToUpdate[53] := "IOVEC_FROMPLC2".O_PRESSLOW;
   #ValuesToUpdate[54] := "IOVEC_FROMPLC2".O_PRESSHIG;
   #ValuesToUpdate[55] := "IOVEC_FROMPLC2".O_ARMHIG;
   #ValuesToUpdate[56] := "IOVEC_FROMPLC2".O_VACON;
   #ValuesToUpdate[57] := "IOVEC_FROMPLC2".O_ARMEXT;
   #ValuesToUpdate[58] := "IOVEC_FROMPLC2".O_ARMCCW;
   #ValuesToUpdate[59] := "IOVEC_FROMPLC2".O_ARMCW;
   #ValuesToUpdate[60] := "IOVEC_FROMPLC2".O_SUEXT;
   #ValuesToUpdate[61] := "IOVEC_FROMPLC2".O_SUUP;
   #ValuesToUpdate[62] := "IOVEC_FROMPLC2".O_SUDWN;
   #ValuesToUpdate[63] := "IOVEC_FROMPLC2".O_SURIGHT;
   #ValuesToUpdate[64] := "IOVEC_FROMPLC2".O_SULEFT;
END_REGION
END_FUNCTION

FUNCTION "putIntDataStruct" : Void   // FC8, LAD
{ S7_Optimized_Access := 'TRUE' }
VERSION : 0.1
   VAR_IN_OUT
      iovec : Array[*] of Bool;
   END_VAR
BEGIN

REGION Network 1 (SCL)
   "DATALOGDATA".Data.I_MAG1EXT := #iovec[0];
   "DATALOGDATA".Data.I_MAG1RET := #iovec[1];
   "DATALOGDATA".Data.I_MAG1EMPT := #iovec[2];
   "DATALOGDATA".Data.I_MAG2EXT := #iovec[3];
   "DATALOGDATA".Data.I_MAG2RET := #iovec[4];
   "DATALOGDATA".Data.I_MAG2EMPT := #iovec[5];
   "DATALOGDATA".Data.I_PSLD := #iovec[6];
   "DATALOGDATA".Data.I_PSCD := #iovec[7];
   "DATALOGDATA".Data.I_PSRD := #iovec[8];
   "DATALOGDATA".Data.I_RELAY1 := #iovec[9];
   "DATALOGDATA".Data.I_LDCEXT := #iovec[10];
   "DATALOGDATA".Data.I_LDCRET := #iovec[11];
   "DATALOGDATA".Data.I_CDCEXT := #iovec[12];
   "DATALOGDATA".Data.I_CDCRET := #iovec[13];
   "DATALOGDATA".Data.I_RDCEXT := #iovec[14];
   "DATALOGDATA".Data.I_RDCRET := #iovec[15];
   "DATALOGDATA".Data.I_WHIT := #iovec[16];
   "DATALOGDATA".Data.I_METAL := #iovec[17];
   "DATALOGDATA".Data.I_PSEOC := #iovec[18];
   "DATALOGDATA".Data.ConcDWN := #iovec[19];
   "DATALOGDATA".Data.ConcUP := #iovec[20];
   "DATALOGDATA".Data.O_MAG1EXT := #iovec[21];
   "DATALOGDATA".Data.O_MAG1RET := #iovec[22];
   "DATALOGDATA".Data.O_MAG2EXT := #iovec[23];
   "DATALOGDATA".Data.O_MAG2RET := #iovec[24];
   "DATALOGDATA".Data.O_RDCEXT := #iovec[25];
   "DATALOGDATA".Data.O_CDCEXT := #iovec[26];
   "DATALOGDATA".Data.O_LDCEXT := #iovec[27];
   "DATALOGDATA".Data.O_CBFW := #iovec[28];
   "DATALOGDATA".Data.O_CBREV := #iovec[29];
   "DATALOGDATA".Data.I_SDO := #iovec[30];
   "DATALOGDATA".Data.I_SDC := #iovec[31];
   "DATALOGDATA".Data.I_AUHEXT := #iovec[32];
   "DATALOGDATA".Data.I_AUHRET := #iovec[33];
   "DATALOGDATA".Data.I_INDARM := #iovec[34];
   "DATALOGDATA".Data.I_ARMLOW := #iovec[35];
   "DATALOGDATA".Data.I_ARMHIG := #iovec[36];
   "DATALOGDATA".Data.I_ARMRET := #iovec[37];
   "DATALOGDATA".Data.I_ARMEXT := #iovec[38];
   "DATALOGDATA".Data.I_SUVE := #iovec[39];
   "DATALOGDATA".Data.I_SUILS := #iovec[40];
   "DATALOGDATA".Data.I_SUSLS := #iovec[41];
   "DATALOGDATA".Data.I_SUEXT := #iovec[42];
   "DATALOGDATA".Data.I_SURET := #iovec[43];
   "DATALOGDATA".Data.I_RELAY2 := #iovec[44];
   "DATALOGDATA".Data.I_SUHE := #iovec[45];
   "DATALOGDATA".Data.I_SURLS := #iovec[46];
   "DATALOGDATA".Data.I_SULLS := #iovec[47];
   "DATALOGDATA".Data.I_SUARMALE := #iovec[48];
   "DATALOGDATA".Data.O_SDO := #iovec[49];
   "DATALOGDATA".Data.O_SDC := #iovec[50];
   "DATALOGDATA".Data.O_AUHRET := #iovec[51];
   "DATALOGDATA".Data.O_AUHEXT := #iovec[52];
   "DATALOGDATA".Data.O_PRESSLOW := #iovec[53];
   "DATALOGDATA".Data.O_PRESSHIG := #iovec[54];
   "DATALOGDATA".Data.O_ARMHIG := #iovec[55];
   "DATALOGDATA".Data.O_VACON := #iovec[56];
   "DATALOGDATA".Data.O_ARMEXT := #iovec[57];
   "DATALOGDATA".Data.O_ARMCCW := #iovec[58];
   "DATALOGDATA".Data.O_ARMCW := #iovec[59];
   "DATALOGDATA".Data.O_SUEXT := #iovec[60];
   "DATALOGDATA".Data.O_SUUP := #iovec[61];
   "DATALOGDATA".Data.O_SUDWN := #iovec[62];
   "DATALOGDATA".Data.O_SURIGHT := #iovec[63];
   "DATALOGDATA".Data.O_SULEFT := #iovec[64];
END_REGION
END_FUNCTION

// folder: Logging/utils

FUNCTION "CompareArrays" : Void   // FC7, LAD
{ S7_Optimized_Access := 'TRUE' }
VERSION : 0.1
   VAR_INPUT
      INPUT1 : Array[*] of Bool;
      INPUT2 : Array[*] of Bool;
   END_VAR
   VAR_TEMP
      out : Bool;
      i : Int;
      dataheaderslowerbound : DInt;
      dataheadersupperbound : DInt;
   END_VAR
BEGIN

REGION Network 1 (SCL)
   #out := TRUE;

   #dataheaderslowerbound := LOWER_BOUND(ARR := #INPUT1, DIM := 1);
   #dataheadersupperbound := UPPER_BOUND(ARR := #INPUT1, DIM := 1);

   FOR #i := #dataheaderslowerbound TO #dataheadersupperbound DO
       // Statement section FOR
       #out := #out AND (#INPUT1[#i] = #INPUT2[#i]);

   END_FOR;

   ENO := NOT #out;
END_REGION
END_FUNCTION

// folder: PetriNet

FUNCTION "ExternalEvents" : Void   // FC1, LAD
{ S7_Optimized_Access := 'TRUE' }
VERSION : 0.1
   VAR_TEMP   // added for the SCL form of the ladder/FBD networks
      _w1 : Bool;
   END_VAR
BEGIN

REGION Network 1: Proximity Sensor End of Conveyor Raising Edge
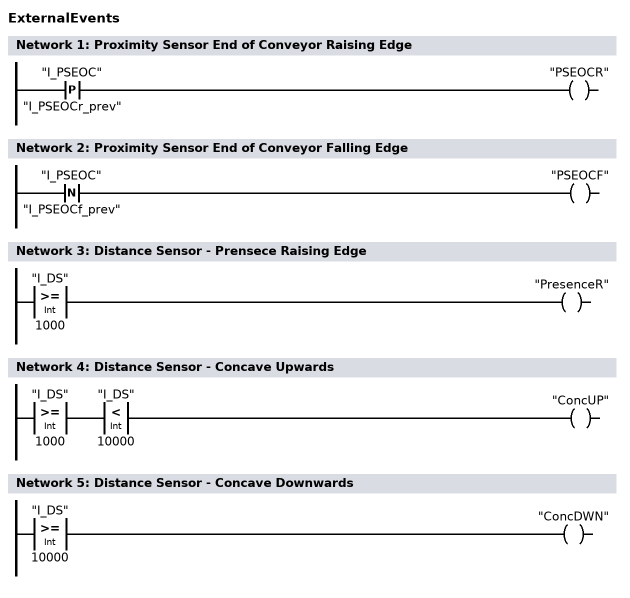
   RUNG wire#powerrail
      P_Contact(operand := "I_PSEOC", bit := "I_PSEOCr_prev")
      Coil( "PSEOCR" )
   END_RUNG
   // the same network as SCL:
   #_w1 := "I_PSEOC" AND NOT "I_PSEOCr_prev";   // rising edge of "I_PSEOC"
   "I_PSEOCr_prev" := "I_PSEOC";
   "PSEOCR" := #_w1;
END_REGION

REGION Network 2: Proximity Sensor End of Conveyor Falling Edge
   RUNG wire#powerrail
      N_Contact(operand := "I_PSEOC", bit := "I_PSEOCf_prev")
      Coil( "PSEOCF" )
   END_RUNG
   // the same network as SCL:
   #_w1 := NOT "I_PSEOC" AND "I_PSEOCf_prev";   // falling edge of "I_PSEOC"
   "I_PSEOCf_prev" := "I_PSEOC";
   "PSEOCF" := #_w1;
END_REGION

REGION Network 3: Distance Sensor - Prensece Raising Edge
   RUNG wire#powerrail
      { S7_Templates := "SrcType := Int" } GE_Contact(in1 := "I_DS", in2 := 1000)
      Coil( "PresenceR" )
   END_RUNG
   // the same network as SCL:
   "PresenceR" := "I_DS" >= 1000;
END_REGION

REGION Network 4: Distance Sensor - Concave Upwards
   RUNG wire#powerrail
      { S7_Templates := "SrcType := Int" } GE_Contact(in1 := "I_DS", in2 := 1000)
      { S7_Templates := "SrcType := Int" } LT_Contact(in1 := "I_DS", in2 := 10000)
      Coil( "ConcUP" )
   END_RUNG
   // the same network as SCL:
   "ConcUP" := ("I_DS" >= 1000) AND ("I_DS" < 10000);
END_REGION

REGION Network 5: Distance Sensor - Concave Downwards
   RUNG wire#powerrail
      { S7_Templates := "SrcType := Int" } GE_Contact(in1 := "I_DS", in2 := 10000)
      Coil( "ConcDWN" )
   END_RUNG
   // the same network as SCL:
   "ConcDWN" := "I_DS" >= 10000;
END_REGION
END_FUNCTION

FUNCTION "Conditions" : Void   // FC2, LAD
{ S7_Optimized_Access := 'TRUE' }
VERSION : 0.1
BEGIN

REGION Network 1: Initialization
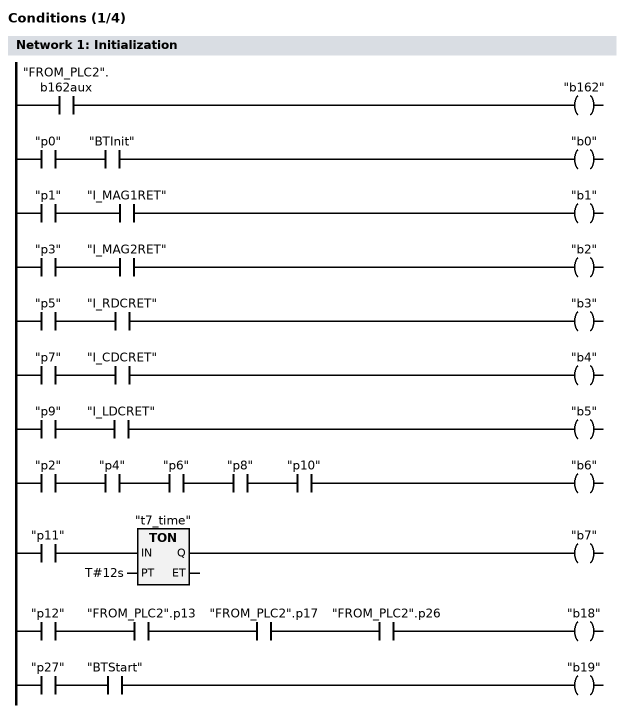
   "b162" := "FROM_PLC2".b162aux;
   "b0" := "p0" AND "BTInit";
   "b1" := "p1" AND "I_MAG1RET";
   "b2" := "p3" AND "I_MAG2RET";
   "b3" := "p5" AND "I_RDCRET";
   "b4" := "p7" AND "I_CDCRET";
   "b5" := "p9" AND "I_LDCRET";
   "b6" := "p2" AND "p4" AND "p6" AND "p8" AND "p10";
   "t7_time".TON(IN := "p11", PT := T#12s);
   "b7" := "t7_time".Q;
   "b18" := "p12" AND "FROM_PLC2".p13 AND "FROM_PLC2".p17 AND "FROM_PLC2".p26;
   "b19" := "p27" AND "BTStart";
END_REGION

REGION Network 2: metalv
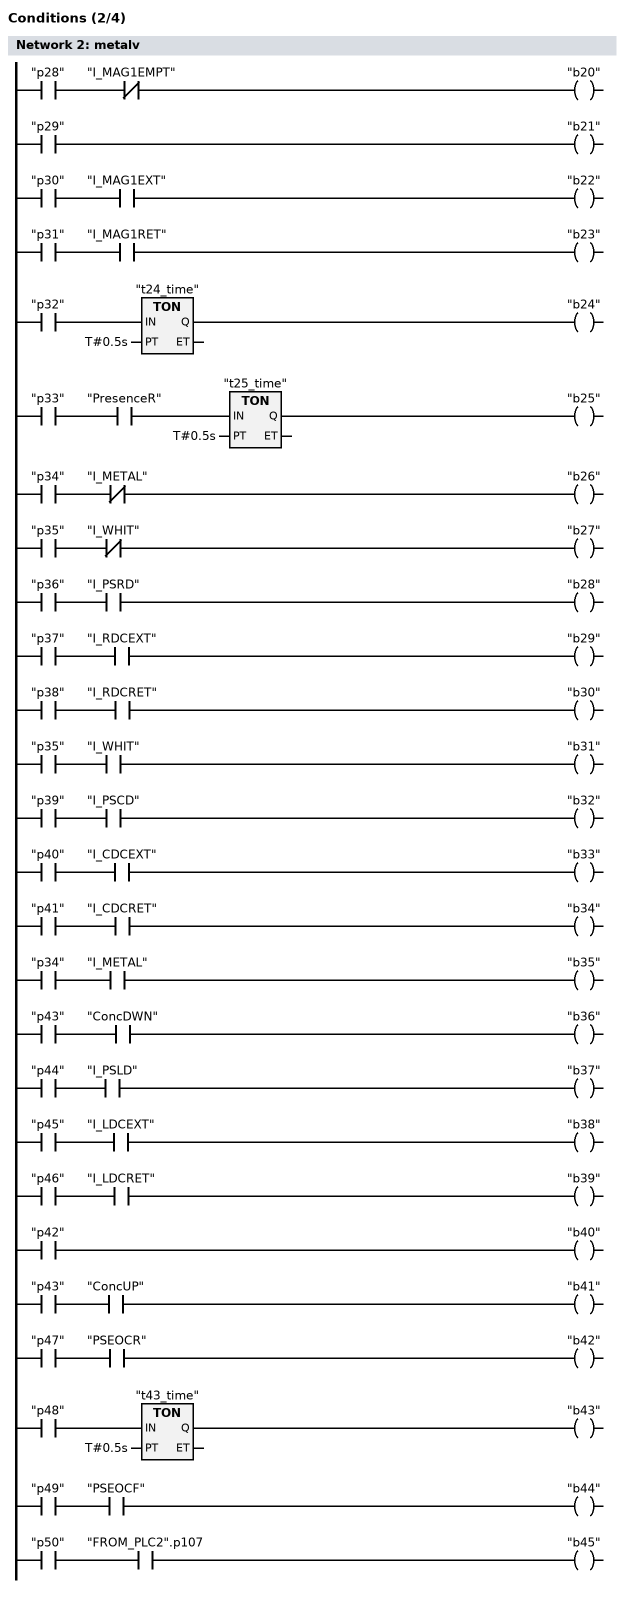
   "b20" := "p28" AND NOT "I_MAG1EMPT";
   "b21" := "p29";
   "b22" := "p30" AND "I_MAG1EXT";
   "b23" := "p31" AND "I_MAG1RET";
   "t24_time".TON(IN := "p32", PT := T#0.5s);
   "b24" := "t24_time".Q;
   "t25_time".TON(IN := "p33" AND "PresenceR", PT := T#0.5s);
   "b25" := "t25_time".Q;
   "b26" := "p34" AND NOT "I_METAL";
   "b27" := "p35" AND NOT "I_WHIT";
   "b28" := "p36" AND "I_PSRD";
   "b29" := "p37" AND "I_RDCEXT";
   "b30" := "p38" AND "I_RDCRET";
   "b31" := "p35" AND "I_WHIT";
   "b32" := "p39" AND "I_PSCD";
   "b33" := "p40" AND "I_CDCEXT";
   "b34" := "p41" AND "I_CDCRET";
   "b35" := "p34" AND "I_METAL";
   "b36" := "p43" AND "ConcDWN";
   "b37" := "p44" AND "I_PSLD";
   "b38" := "p45" AND "I_LDCEXT";
   "b39" := "p46" AND "I_LDCRET";
   "b40" := "p42";
   "b41" := "p43" AND "ConcUP";
   "b42" := "p47" AND "PSEOCR";
   "t43_time".TON(IN := "p48", PT := T#0.5s);
   "b43" := "t43_time".Q;
   "b44" := "p49" AND "PSEOCF";
   "b45" := "p50" AND "FROM_PLC2".p107;
END_REGION

REGION Network 3: plastic
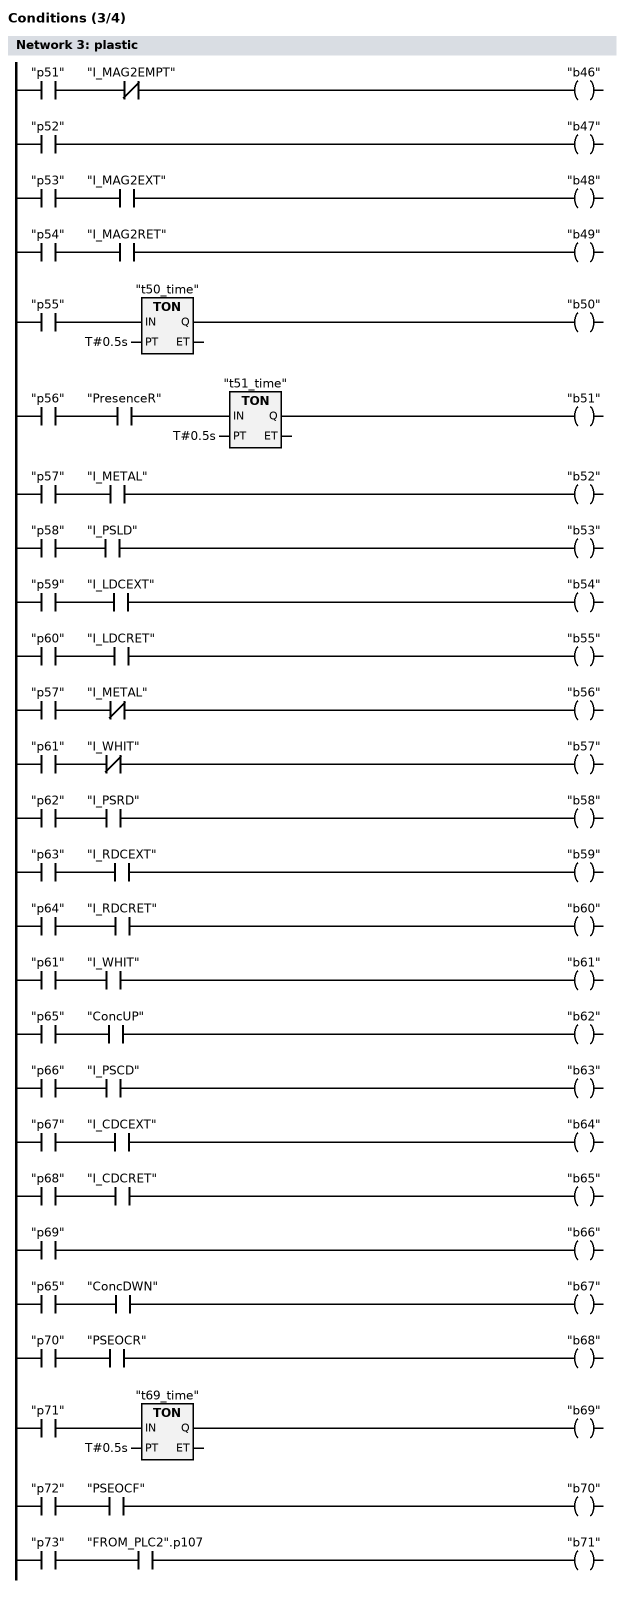
   "b46" := "p51" AND NOT "I_MAG2EMPT";
   "b47" := "p52";
   "b48" := "p53" AND "I_MAG2EXT";
   "b49" := "p54" AND "I_MAG2RET";
   "t50_time".TON(IN := "p55", PT := T#0.5s);
   "b50" := "t50_time".Q;
   "t51_time".TON(IN := "p56" AND "PresenceR", PT := T#0.5s);
   "b51" := "t51_time".Q;
   "b52" := "p57" AND "I_METAL";
   "b53" := "p58" AND "I_PSLD";
   "b54" := "p59" AND "I_LDCEXT";
   "b55" := "p60" AND "I_LDCRET";
   "b56" := "p57" AND NOT "I_METAL";
   "b57" := "p61" AND NOT "I_WHIT";
   "b58" := "p62" AND "I_PSRD";
   "b59" := "p63" AND "I_RDCEXT";
   "b60" := "p64" AND "I_RDCRET";
   "b61" := "p61" AND "I_WHIT";
   "b62" := "p65" AND "ConcUP";
   "b63" := "p66" AND "I_PSCD";
   "b64" := "p67" AND "I_CDCEXT";
   "b65" := "p68" AND "I_CDCRET";
   "b66" := "p69";
   "b67" := "p65" AND "ConcDWN";
   "b68" := "p70" AND "PSEOCR";
   "t69_time".TON(IN := "p71", PT := T#0.5s);
   "b69" := "t69_time".Q;
   "b70" := "p72" AND "PSEOCF";
   "b71" := "p73" AND "FROM_PLC2".p107;
END_REGION

REGION Network 4: Arm Stop
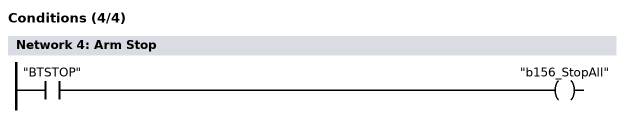
   RUNG wire#powerrail
      Contact( "BTSTOP" )
      Coil( "b156_StopAll" )
   END_RUNG
   // the same network as SCL:
   "b156_StopAll" := "BTSTOP";
END_REGION
END_FUNCTION

FUNCTION "Dynamics" : Void   // FC3, LAD
{ S7_Optimized_Access := 'TRUE' }
VERSION : 0.1
BEGIN

REGION Network 1: Initialization
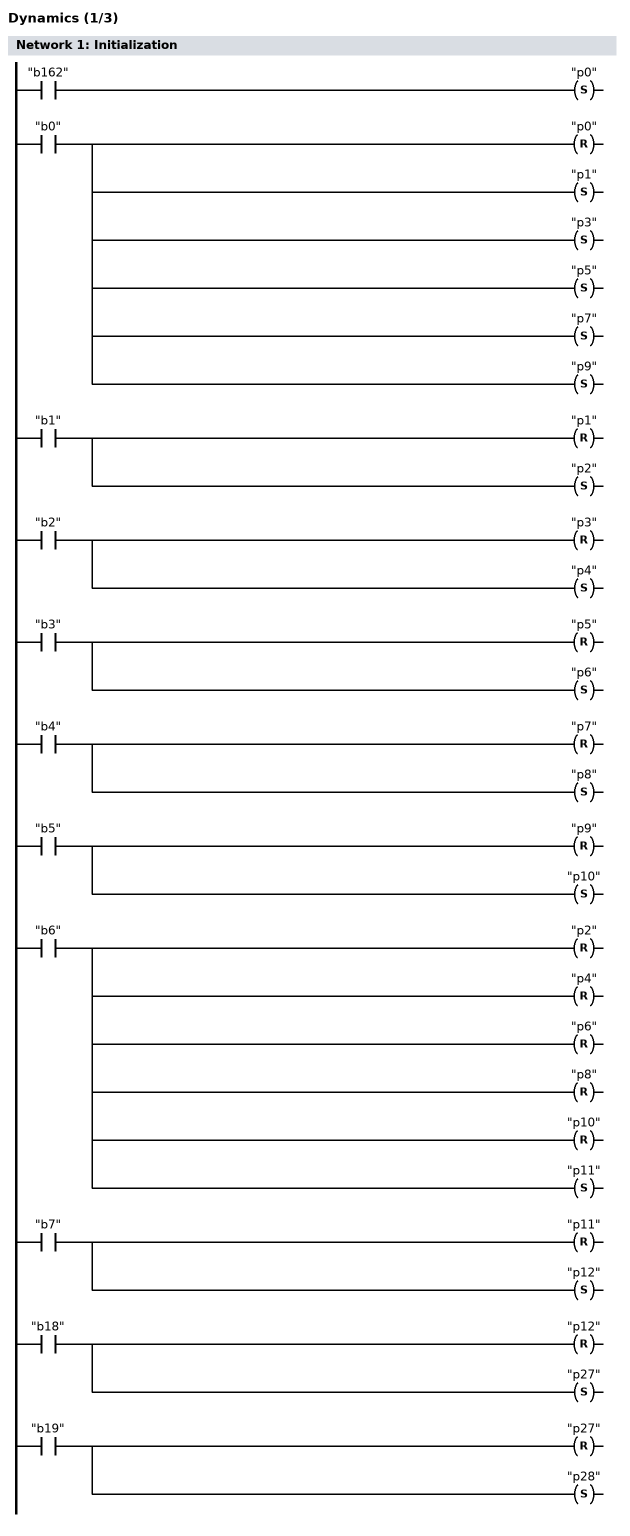
   RUNG wire#powerrail
      Contact( "b162" )
      S_Coil( "p0" )
   END_RUNG
   RUNG wire#powerrail
      Contact( "b0" )
      wire#w1
      R_Coil( "p0" )
   END_RUNG
   RUNG wire#w1
      S_Coil( "p1" )
   END_RUNG
   RUNG wire#w1
      S_Coil( "p3" )
   END_RUNG
   RUNG wire#w1
      S_Coil( "p5" )
   END_RUNG
   RUNG wire#w1
      S_Coil( "p7" )
   END_RUNG
   RUNG wire#w1
      S_Coil( "p9" )
   END_RUNG
   RUNG wire#powerrail
      Contact( "b1" )
      wire#w2
      R_Coil( "p1" )
   END_RUNG
   RUNG wire#w2
      S_Coil( "p2" )
   END_RUNG
   RUNG wire#powerrail
      Contact( "b2" )
      wire#w3
      R_Coil( "p3" )
   END_RUNG
   RUNG wire#w3
      S_Coil( "p4" )
   END_RUNG
   RUNG wire#powerrail
      Contact( "b3" )
      wire#w4
      R_Coil( "p5" )
   END_RUNG
   RUNG wire#w4
      S_Coil( "p6" )
   END_RUNG
   RUNG wire#powerrail
      Contact( "b4" )
      wire#w5
      R_Coil( "p7" )
   END_RUNG
   RUNG wire#w5
      S_Coil( "p8" )
   END_RUNG
   RUNG wire#powerrail
      Contact( "b5" )
      wire#w6
      R_Coil( "p9" )
   END_RUNG
   RUNG wire#w6
      S_Coil( "p10" )
   END_RUNG
   RUNG wire#powerrail
      Contact( "b6" )
      wire#w7
      R_Coil( "p2" )
   END_RUNG
   RUNG wire#w7
      R_Coil( "p4" )
   END_RUNG
   RUNG wire#w7
      R_Coil( "p6" )
   END_RUNG
   RUNG wire#w7
      R_Coil( "p8" )
   END_RUNG
   RUNG wire#w7
      R_Coil( "p10" )
   END_RUNG
   RUNG wire#w7
      S_Coil( "p11" )
   END_RUNG
   RUNG wire#powerrail
      Contact( "b7" )
      wire#w8
      R_Coil( "p11" )
   END_RUNG
   RUNG wire#w8
      S_Coil( "p12" )
   END_RUNG
   RUNG wire#powerrail
      Contact( "b18" )
      wire#w9
      R_Coil( "p12" )
   END_RUNG
   RUNG wire#w9
      S_Coil( "p27" )
   END_RUNG
   RUNG wire#powerrail
      Contact( "b19" )
      wire#w10
      R_Coil( "p27" )
   END_RUNG
   RUNG wire#w10
      S_Coil( "p28" )
   END_RUNG
   // the same network as SCL:
   IF "b162" THEN "p0" := TRUE; END_IF;
   IF "b0" THEN
       "p0" := FALSE;
       "p1" := TRUE;
       "p3" := TRUE;
       "p5" := TRUE;
       "p7" := TRUE;
       "p9" := TRUE;
   END_IF;
   IF "b1" THEN
       "p1" := FALSE;
       "p2" := TRUE;
   END_IF;
   IF "b2" THEN
       "p3" := FALSE;
       "p4" := TRUE;
   END_IF;
   IF "b3" THEN
       "p5" := FALSE;
       "p6" := TRUE;
   END_IF;
   IF "b4" THEN
       "p7" := FALSE;
       "p8" := TRUE;
   END_IF;
   IF "b5" THEN
       "p9" := FALSE;
       "p10" := TRUE;
   END_IF;
   IF "b6" THEN
       "p2" := FALSE;
       "p4" := FALSE;
       "p6" := FALSE;
       "p8" := FALSE;
       "p10" := FALSE;
       "p11" := TRUE;
   END_IF;
   IF "b7" THEN
       "p11" := FALSE;
       "p12" := TRUE;
   END_IF;
   IF "b18" THEN
       "p12" := FALSE;
       "p27" := TRUE;
   END_IF;
   IF "b19" THEN
       "p27" := FALSE;
       "p28" := TRUE;
   END_IF;
END_REGION

REGION Network 2: metal v
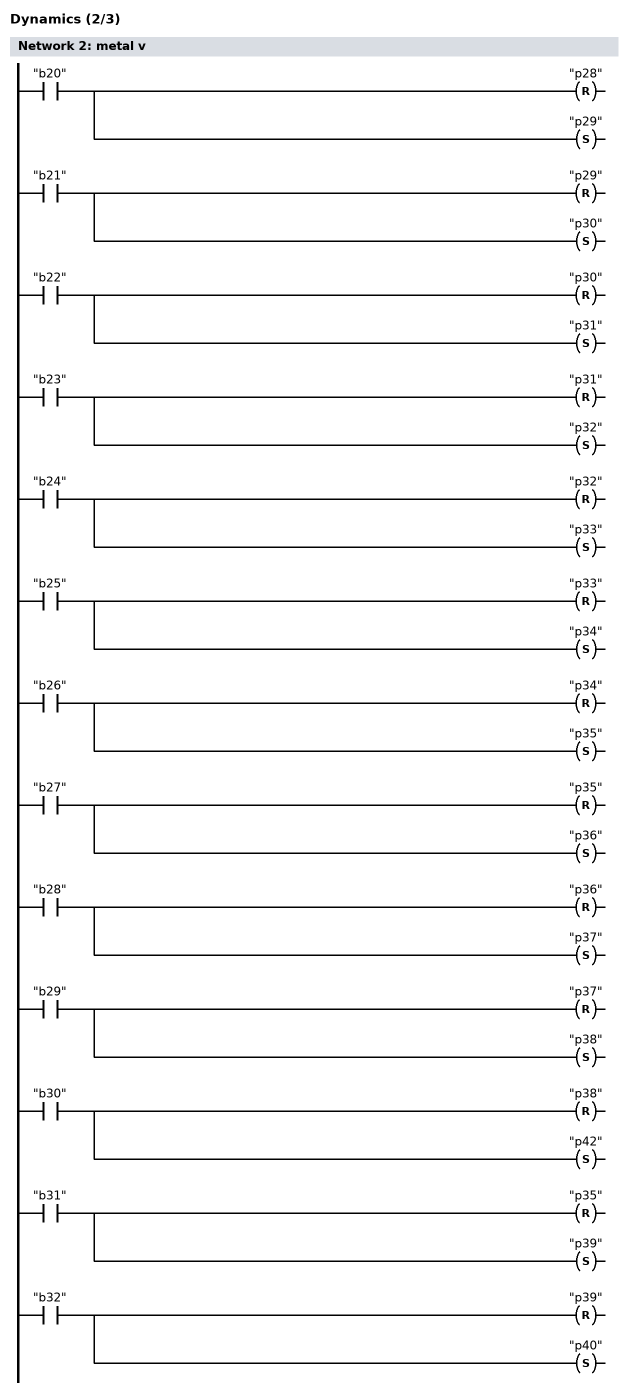
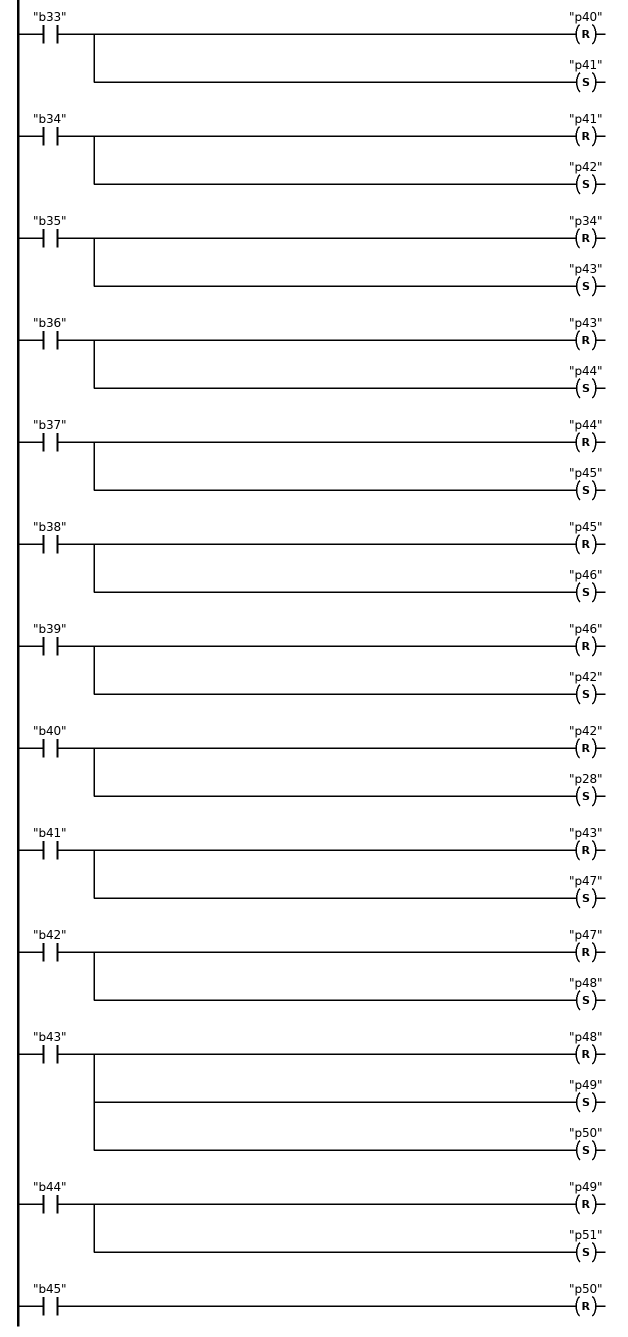
   RUNG wire#powerrail
      Contact( "b20" )
      wire#w1
      R_Coil( "p28" )
   END_RUNG
   RUNG wire#w1
      S_Coil( "p29" )
   END_RUNG
   RUNG wire#powerrail
      Contact( "b21" )
      wire#w2
      R_Coil( "p29" )
   END_RUNG
   RUNG wire#w2
      S_Coil( "p30" )
   END_RUNG
   RUNG wire#powerrail
      Contact( "b22" )
      wire#w3
      R_Coil( "p30" )
   END_RUNG
   RUNG wire#w3
      S_Coil( "p31" )
   END_RUNG
   RUNG wire#powerrail
      Contact( "b23" )
      wire#w4
      R_Coil( "p31" )
   END_RUNG
   RUNG wire#w4
      S_Coil( "p32" )
   END_RUNG
   RUNG wire#powerrail
      Contact( "b24" )
      wire#w5
      R_Coil( "p32" )
   END_RUNG
   RUNG wire#w5
      S_Coil( "p33" )
   END_RUNG
   RUNG wire#powerrail
      Contact( "b25" )
      wire#w6
      R_Coil( "p33" )
   END_RUNG
   RUNG wire#w6
      S_Coil( "p34" )
   END_RUNG
   RUNG wire#powerrail
      Contact( "b26" )
      wire#w7
      R_Coil( "p34" )
   END_RUNG
   RUNG wire#w7
      S_Coil( "p35" )
   END_RUNG
   RUNG wire#powerrail
      Contact( "b27" )
      wire#w8
      R_Coil( "p35" )
   END_RUNG
   RUNG wire#w8
      S_Coil( "p36" )
   END_RUNG
   RUNG wire#powerrail
      Contact( "b28" )
      wire#w9
      R_Coil( "p36" )
   END_RUNG
   RUNG wire#w9
      S_Coil( "p37" )
   END_RUNG
   RUNG wire#powerrail
      Contact( "b29" )
      wire#w10
      R_Coil( "p37" )
   END_RUNG
   RUNG wire#w10
      S_Coil( "p38" )
   END_RUNG
   RUNG wire#powerrail
      Contact( "b30" )
      wire#w11
      R_Coil( "p38" )
   END_RUNG
   RUNG wire#w11
      S_Coil( "p42" )
   END_RUNG
   RUNG wire#powerrail
      Contact( "b31" )
      wire#w12
      R_Coil( "p35" )
   END_RUNG
   RUNG wire#w12
      S_Coil( "p39" )
   END_RUNG
   RUNG wire#powerrail
      Contact( "b32" )
      wire#w13
      R_Coil( "p39" )
   END_RUNG
   RUNG wire#w13
      S_Coil( "p40" )
   END_RUNG
   RUNG wire#powerrail
      Contact( "b33" )
      wire#w14
      R_Coil( "p40" )
   END_RUNG
   RUNG wire#w14
      S_Coil( "p41" )
   END_RUNG
   RUNG wire#powerrail
      Contact( "b34" )
      wire#w15
      R_Coil( "p41" )
   END_RUNG
   RUNG wire#w15
      S_Coil( "p42" )
   END_RUNG
   RUNG wire#powerrail
      Contact( "b35" )
      wire#w16
      R_Coil( "p34" )
   END_RUNG
   RUNG wire#w16
      S_Coil( "p43" )
   END_RUNG
   RUNG wire#powerrail
      Contact( "b36" )
      wire#w17
      R_Coil( "p43" )
   END_RUNG
   RUNG wire#w17
      S_Coil( "p44" )
   END_RUNG
   RUNG wire#powerrail
      Contact( "b37" )
      wire#w18
      R_Coil( "p44" )
   END_RUNG
   RUNG wire#w18
      S_Coil( "p45" )
   END_RUNG
   RUNG wire#powerrail
      Contact( "b38" )
      wire#w19
      R_Coil( "p45" )
   END_RUNG
   RUNG wire#w19
      S_Coil( "p46" )
   END_RUNG
   RUNG wire#powerrail
      Contact( "b39" )
      wire#w20
      R_Coil( "p46" )
   END_RUNG
   RUNG wire#w20
      S_Coil( "p42" )
   END_RUNG
   RUNG wire#powerrail
      Contact( "b40" )
      wire#w21
      R_Coil( "p42" )
   END_RUNG
   RUNG wire#w21
      S_Coil( "p28" )
   END_RUNG
   RUNG wire#powerrail
      Contact( "b41" )
      wire#w22
      R_Coil( "p43" )
   END_RUNG
   RUNG wire#w22
      S_Coil( "p47" )
   END_RUNG
   RUNG wire#powerrail
      Contact( "b42" )
      wire#w23
      R_Coil( "p47" )
   END_RUNG
   RUNG wire#w23
      S_Coil( "p48" )
   END_RUNG
   RUNG wire#powerrail
      Contact( "b43" )
      wire#w24
      R_Coil( "p48" )
   END_RUNG
   RUNG wire#w24
      S_Coil( "p49" )
   END_RUNG
   RUNG wire#w24
      S_Coil( "p50" )
   END_RUNG
   RUNG wire#powerrail
      Contact( "b44" )
      wire#w25
      R_Coil( "p49" )
   END_RUNG
   RUNG wire#w25
      S_Coil( "p51" )
   END_RUNG
   RUNG wire#powerrail
      Contact( "b45" )
      R_Coil( "p50" )
   END_RUNG
   // the same network as SCL:
   IF "b20" THEN
       "p28" := FALSE;
       "p29" := TRUE;
   END_IF;
   IF "b21" THEN
       "p29" := FALSE;
       "p30" := TRUE;
   END_IF;
   IF "b22" THEN
       "p30" := FALSE;
       "p31" := TRUE;
   END_IF;
   IF "b23" THEN
       "p31" := FALSE;
       "p32" := TRUE;
   END_IF;
   IF "b24" THEN
       "p32" := FALSE;
       "p33" := TRUE;
   END_IF;
   IF "b25" THEN
       "p33" := FALSE;
       "p34" := TRUE;
   END_IF;
   IF "b26" THEN
       "p34" := FALSE;
       "p35" := TRUE;
   END_IF;
   IF "b27" THEN
       "p35" := FALSE;
       "p36" := TRUE;
   END_IF;
   IF "b28" THEN
       "p36" := FALSE;
       "p37" := TRUE;
   END_IF;
   IF "b29" THEN
       "p37" := FALSE;
       "p38" := TRUE;
   END_IF;
   IF "b30" THEN
       "p38" := FALSE;
       "p42" := TRUE;
   END_IF;
   IF "b31" THEN
       "p35" := FALSE;
       "p39" := TRUE;
   END_IF;
   IF "b32" THEN
       "p39" := FALSE;
       "p40" := TRUE;
   END_IF;
   IF "b33" THEN
       "p40" := FALSE;
       "p41" := TRUE;
   END_IF;
   IF "b34" THEN
       "p41" := FALSE;
       "p42" := TRUE;
   END_IF;
   IF "b35" THEN
       "p34" := FALSE;
       "p43" := TRUE;
   END_IF;
   IF "b36" THEN
       "p43" := FALSE;
       "p44" := TRUE;
   END_IF;
   IF "b37" THEN
       "p44" := FALSE;
       "p45" := TRUE;
   END_IF;
   IF "b38" THEN
       "p45" := FALSE;
       "p46" := TRUE;
   END_IF;
   IF "b39" THEN
       "p46" := FALSE;
       "p42" := TRUE;
   END_IF;
   IF "b40" THEN
       "p42" := FALSE;
       "p28" := TRUE;
   END_IF;
   IF "b41" THEN
       "p43" := FALSE;
       "p47" := TRUE;
   END_IF;
   IF "b42" THEN
       "p47" := FALSE;
       "p48" := TRUE;
   END_IF;
   IF "b43" THEN
       "p48" := FALSE;
       "p49" := TRUE;
       "p50" := TRUE;
   END_IF;
   IF "b44" THEN
       "p49" := FALSE;
       "p51" := TRUE;
   END_IF;
   IF "b45" THEN "p50" := FALSE; END_IF;
END_REGION

REGION Network 3: plastic ^
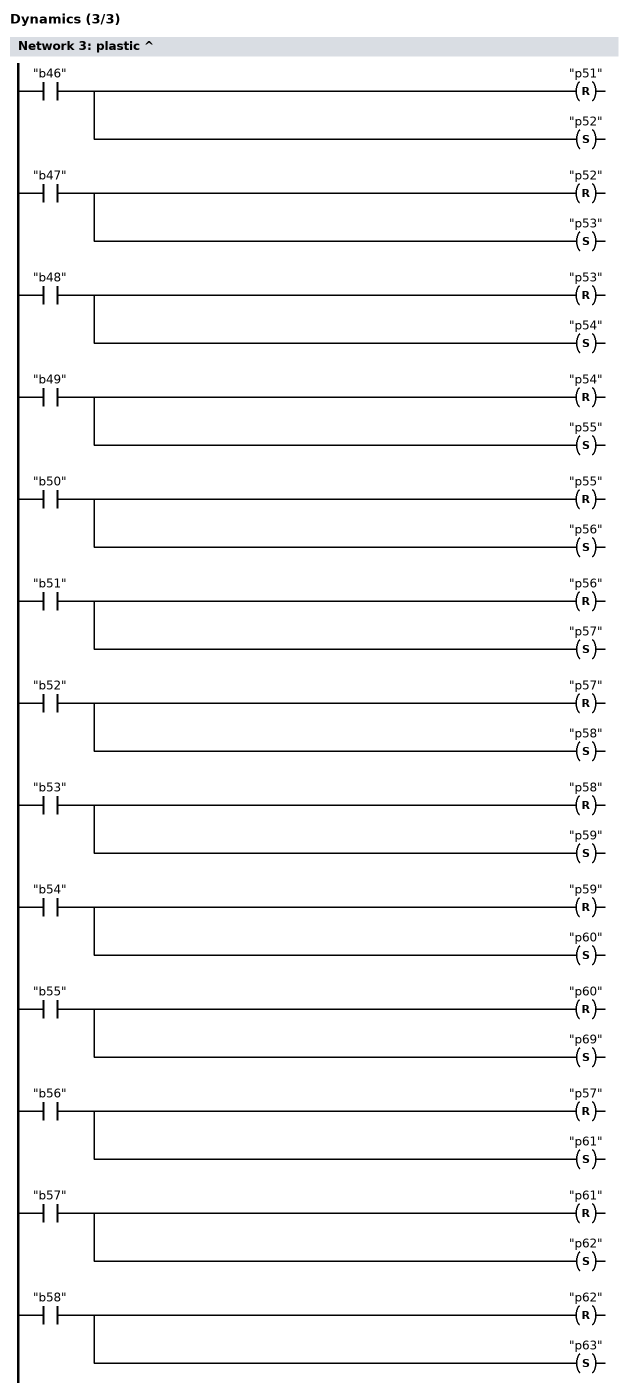
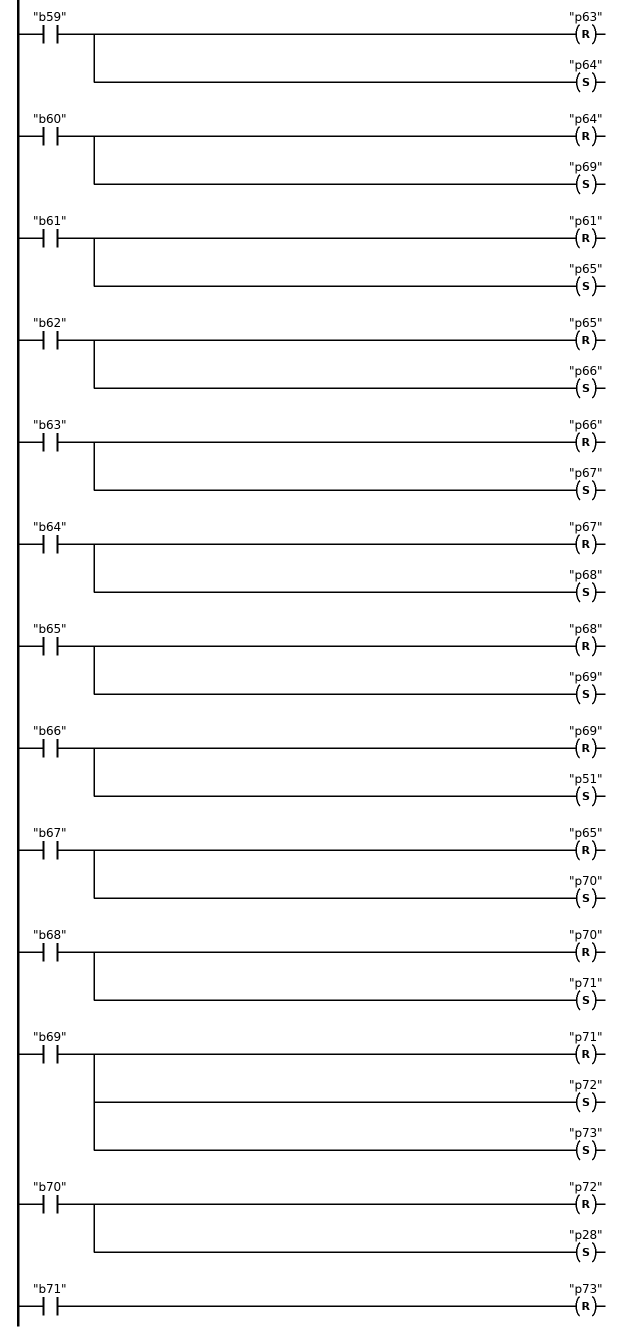
   RUNG wire#powerrail
      Contact( "b46" )
      wire#w1
      R_Coil( "p51" )
   END_RUNG
   RUNG wire#w1
      S_Coil( "p52" )
   END_RUNG
   RUNG wire#powerrail
      Contact( "b47" )
      wire#w2
      R_Coil( "p52" )
   END_RUNG
   RUNG wire#w2
      S_Coil( "p53" )
   END_RUNG
   RUNG wire#powerrail
      Contact( "b48" )
      wire#w3
      R_Coil( "p53" )
   END_RUNG
   RUNG wire#w3
      S_Coil( "p54" )
   END_RUNG
   RUNG wire#powerrail
      Contact( "b49" )
      wire#w4
      R_Coil( "p54" )
   END_RUNG
   RUNG wire#w4
      S_Coil( "p55" )
   END_RUNG
   RUNG wire#powerrail
      Contact( "b50" )
      wire#w5
      R_Coil( "p55" )
   END_RUNG
   RUNG wire#w5
      S_Coil( "p56" )
   END_RUNG
   RUNG wire#powerrail
      Contact( "b51" )
      wire#w6
      R_Coil( "p56" )
   END_RUNG
   RUNG wire#w6
      S_Coil( "p57" )
   END_RUNG
   RUNG wire#powerrail
      Contact( "b52" )
      wire#w7
      R_Coil( "p57" )
   END_RUNG
   RUNG wire#w7
      S_Coil( "p58" )
   END_RUNG
   RUNG wire#powerrail
      Contact( "b53" )
      wire#w8
      R_Coil( "p58" )
   END_RUNG
   RUNG wire#w8
      S_Coil( "p59" )
   END_RUNG
   RUNG wire#powerrail
      Contact( "b54" )
      wire#w9
      R_Coil( "p59" )
   END_RUNG
   RUNG wire#w9
      S_Coil( "p60" )
   END_RUNG
   RUNG wire#powerrail
      Contact( "b55" )
      wire#w10
      R_Coil( "p60" )
   END_RUNG
   RUNG wire#w10
      S_Coil( "p69" )
   END_RUNG
   RUNG wire#powerrail
      Contact( "b56" )
      wire#w11
      R_Coil( "p57" )
   END_RUNG
   RUNG wire#w11
      S_Coil( "p61" )
   END_RUNG
   RUNG wire#powerrail
      Contact( "b57" )
      wire#w12
      R_Coil( "p61" )
   END_RUNG
   RUNG wire#w12
      S_Coil( "p62" )
   END_RUNG
   RUNG wire#powerrail
      Contact( "b58" )
      wire#w13
      R_Coil( "p62" )
   END_RUNG
   RUNG wire#w13
      S_Coil( "p63" )
   END_RUNG
   RUNG wire#powerrail
      Contact( "b59" )
      wire#w14
      R_Coil( "p63" )
   END_RUNG
   RUNG wire#w14
      S_Coil( "p64" )
   END_RUNG
   RUNG wire#powerrail
      Contact( "b60" )
      wire#w15
      R_Coil( "p64" )
   END_RUNG
   RUNG wire#w15
      S_Coil( "p69" )
   END_RUNG
   RUNG wire#powerrail
      Contact( "b61" )
      wire#w16
      R_Coil( "p61" )
   END_RUNG
   RUNG wire#w16
      S_Coil( "p65" )
   END_RUNG
   RUNG wire#powerrail
      Contact( "b62" )
      wire#w17
      R_Coil( "p65" )
   END_RUNG
   RUNG wire#w17
      S_Coil( "p66" )
   END_RUNG
   RUNG wire#powerrail
      Contact( "b63" )
      wire#w18
      R_Coil( "p66" )
   END_RUNG
   RUNG wire#w18
      S_Coil( "p67" )
   END_RUNG
   RUNG wire#powerrail
      Contact( "b64" )
      wire#w19
      R_Coil( "p67" )
   END_RUNG
   RUNG wire#w19
      S_Coil( "p68" )
   END_RUNG
   RUNG wire#powerrail
      Contact( "b65" )
      wire#w20
      R_Coil( "p68" )
   END_RUNG
   RUNG wire#w20
      S_Coil( "p69" )
   END_RUNG
   RUNG wire#powerrail
      Contact( "b66" )
      wire#w21
      R_Coil( "p69" )
   END_RUNG
   RUNG wire#w21
      S_Coil( "p51" )
   END_RUNG
   RUNG wire#powerrail
      Contact( "b67" )
      wire#w22
      R_Coil( "p65" )
   END_RUNG
   RUNG wire#w22
      S_Coil( "p70" )
   END_RUNG
   RUNG wire#powerrail
      Contact( "b68" )
      wire#w23
      R_Coil( "p70" )
   END_RUNG
   RUNG wire#w23
      S_Coil( "p71" )
   END_RUNG
   RUNG wire#powerrail
      Contact( "b69" )
      wire#w24
      R_Coil( "p71" )
   END_RUNG
   RUNG wire#w24
      S_Coil( "p72" )
   END_RUNG
   RUNG wire#w24
      S_Coil( "p73" )
   END_RUNG
   RUNG wire#powerrail
      Contact( "b70" )
      wire#w25
      R_Coil( "p72" )
   END_RUNG
   RUNG wire#w25
      S_Coil( "p28" )
   END_RUNG
   RUNG wire#powerrail
      Contact( "b71" )
      R_Coil( "p73" )
   END_RUNG
   // the same network as SCL:
   IF "b46" THEN
       "p51" := FALSE;
       "p52" := TRUE;
   END_IF;
   IF "b47" THEN
       "p52" := FALSE;
       "p53" := TRUE;
   END_IF;
   IF "b48" THEN
       "p53" := FALSE;
       "p54" := TRUE;
   END_IF;
   IF "b49" THEN
       "p54" := FALSE;
       "p55" := TRUE;
   END_IF;
   IF "b50" THEN
       "p55" := FALSE;
       "p56" := TRUE;
   END_IF;
   IF "b51" THEN
       "p56" := FALSE;
       "p57" := TRUE;
   END_IF;
   IF "b52" THEN
       "p57" := FALSE;
       "p58" := TRUE;
   END_IF;
   IF "b53" THEN
       "p58" := FALSE;
       "p59" := TRUE;
   END_IF;
   IF "b54" THEN
       "p59" := FALSE;
       "p60" := TRUE;
   END_IF;
   IF "b55" THEN
       "p60" := FALSE;
       "p69" := TRUE;
   END_IF;
   IF "b56" THEN
       "p57" := FALSE;
       "p61" := TRUE;
   END_IF;
   IF "b57" THEN
       "p61" := FALSE;
       "p62" := TRUE;
   END_IF;
   IF "b58" THEN
       "p62" := FALSE;
       "p63" := TRUE;
   END_IF;
   IF "b59" THEN
       "p63" := FALSE;
       "p64" := TRUE;
   END_IF;
   IF "b60" THEN
       "p64" := FALSE;
       "p69" := TRUE;
   END_IF;
   IF "b61" THEN
       "p61" := FALSE;
       "p65" := TRUE;
   END_IF;
   IF "b62" THEN
       "p65" := FALSE;
       "p66" := TRUE;
   END_IF;
   IF "b63" THEN
       "p66" := FALSE;
       "p67" := TRUE;
   END_IF;
   IF "b64" THEN
       "p67" := FALSE;
       "p68" := TRUE;
   END_IF;
   IF "b65" THEN
       "p68" := FALSE;
       "p69" := TRUE;
   END_IF;
   IF "b66" THEN
       "p69" := FALSE;
       "p51" := TRUE;
   END_IF;
   IF "b67" THEN
       "p65" := FALSE;
       "p70" := TRUE;
   END_IF;
   IF "b68" THEN
       "p70" := FALSE;
       "p71" := TRUE;
   END_IF;
   IF "b69" THEN
       "p71" := FALSE;
       "p72" := TRUE;
       "p73" := TRUE;
   END_IF;
   IF "b70" THEN
       "p72" := FALSE;
       "p28" := TRUE;
   END_IF;
   IF "b71" THEN "p73" := FALSE; END_IF;
END_REGION

REGION Network 4 (SCL): Arm Stop
   IF "b156_StopAll" THEN
       "p1" := 0;
       "p2" := 0;
       "p3" := 0;
       "p4" := 0;
       "p5" := 0;
       "p6" := 0;
       "p7" := 0;
       "p8" := 0;
       "p9" := 0;
       "p10" := 0;
       "p11" := 0;
       "p12" := 0;
       "p27" := 0;
       "p28" := 0;
       "p29" := 0;
       "p30" := 0;
       "p31" := 0;
       "p32" := 0;
       "p33" := 0;
       "p34" := 0;
       "p35" := 0;
       "p36" := 0;
       "p37" := 0;
       "p38" := 0;
       "p39" := 0;
       "p40" := 0;
       "p41" := 0;
       "p42" := 0;
       "p43" := 0;
       "p44" := 0;
       "p45" := 0;
       "p46" := 0;
       "p47" := 0;
       "p48" := 0;
       "p49" := 0;
       "p50" := 0;
       "p51" := 0;
       "p52" := 0;
       "p53" := 0;
       "p54" := 0;
       "p55" := 0;
       "p56" := 0;
       "p57" := 0;
       "p58" := 0;
       "p59" := 0;
       "p60" := 0;
       "p61" := 0;
       "p62" := 0;
       "p63" := 0;
       "p64" := 0;
       "p65" := 0;
       "p66" := 0;
       "p67" := 0;
       "p68" := 0;
       "p69" := 0;
       "p70" := 0;
       "p71" := 0;
       "p72" := 0;
       "p73" := 0;
   END_IF;
END_REGION
END_FUNCTION

FUNCTION "Initialization" : Void   // FC4, LAD
{ S7_Optimized_Access := 'TRUE' }
VERSION : 0.1
BEGIN

REGION Network 1
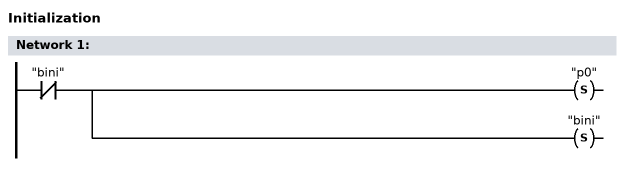
   RUNG wire#powerrail
      I_Contact( "bini" )
      wire#w1
      S_Coil( "p0" )
   END_RUNG
   RUNG wire#w1
      S_Coil( "bini" )
   END_RUNG
   // the same network as SCL:
   IF NOT "bini" THEN
       "p0" := TRUE;
       "bini" := TRUE;
   END_IF;
END_REGION
END_FUNCTION

FUNCTION "Actions" : Void   // FC5, LAD
{ S7_Optimized_Access := 'TRUE' }
VERSION : 0.1
BEGIN

REGION Network 1: Retract MAG 1 Cylinder
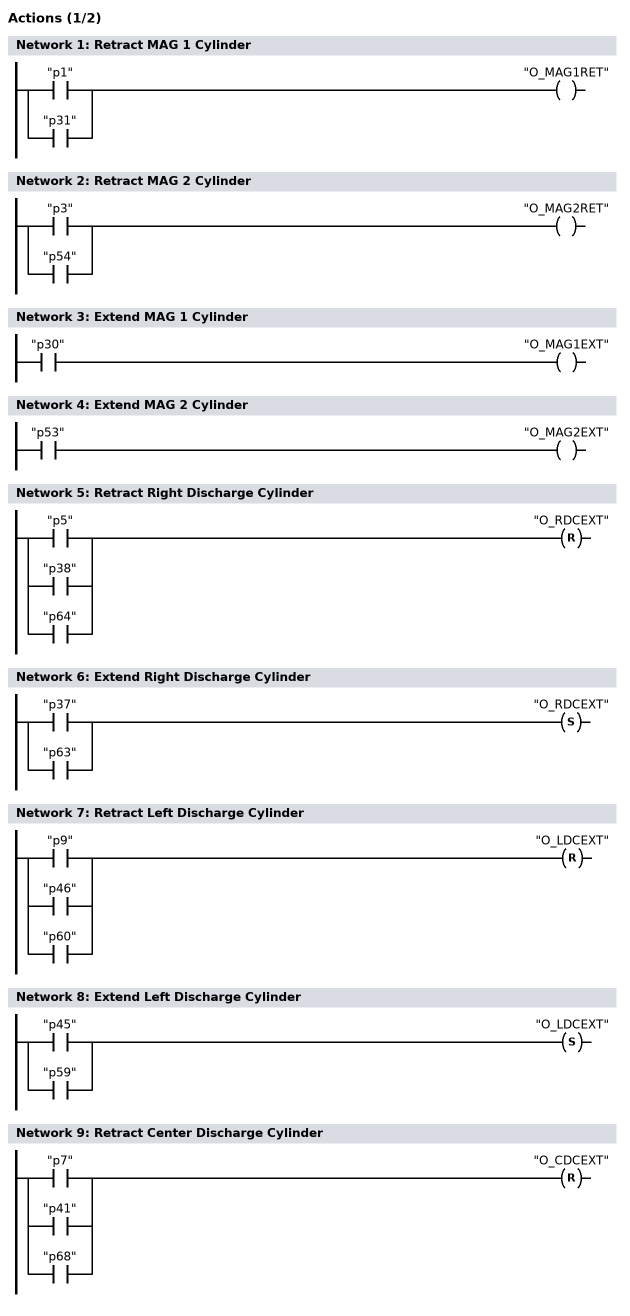
   RUNG wire#powerrail
      Contact( "p1" )
      wire#w1
      Coil( "O_MAG1RET" )
   END_RUNG
   RUNG wire#powerrail
      Contact( "p31" )
   END_RUNG wire#w1
   // the same network as SCL:
   "O_MAG1RET" := "p1" OR "p31";
END_REGION

REGION Network 2: Retract MAG 2 Cylinder
   RUNG wire#powerrail
      Contact( "p3" )
      wire#w1
      Coil( "O_MAG2RET" )
   END_RUNG
   RUNG wire#powerrail
      Contact( "p54" )
   END_RUNG wire#w1
   // the same network as SCL:
   "O_MAG2RET" := "p3" OR "p54";
END_REGION

REGION Network 3: Extend MAG 1 Cylinder
   RUNG wire#powerrail
      Contact( "p30" )
      Coil( "O_MAG1EXT" )
   END_RUNG
   // the same network as SCL:
   "O_MAG1EXT" := "p30";
END_REGION

REGION Network 4: Extend MAG 2 Cylinder
   RUNG wire#powerrail
      Contact( "p53" )
      Coil( "O_MAG2EXT" )
   END_RUNG
   // the same network as SCL:
   "O_MAG2EXT" := "p53";
END_REGION

REGION Network 5: Retract Right Discharge Cylinder
   RUNG wire#powerrail
      Contact( "p5" )
      wire#w1
      R_Coil( "O_RDCEXT" )
   END_RUNG
   RUNG wire#powerrail
      Contact( "p38" )
   END_RUNG wire#w1
   RUNG wire#powerrail
      Contact( "p64" )
   END_RUNG wire#w1
   // the same network as SCL:
   IF "p5" OR "p38" OR "p64" THEN "O_RDCEXT" := FALSE; END_IF;
END_REGION

REGION Network 6: Extend Right Discharge Cylinder
   RUNG wire#powerrail
      Contact( "p37" )
      wire#w1
      S_Coil( "O_RDCEXT" )
   END_RUNG
   RUNG wire#powerrail
      Contact( "p63" )
   END_RUNG wire#w1
   // the same network as SCL:
   IF "p37" OR "p63" THEN "O_RDCEXT" := TRUE; END_IF;
END_REGION

REGION Network 7: Retract Left Discharge Cylinder
   RUNG wire#powerrail
      Contact( "p9" )
      wire#w1
      R_Coil( "O_LDCEXT" )
   END_RUNG
   RUNG wire#powerrail
      Contact( "p46" )
   END_RUNG wire#w1
   RUNG wire#powerrail
      Contact( "p60" )
   END_RUNG wire#w1
   // the same network as SCL:
   IF "p9" OR "p46" OR "p60" THEN "O_LDCEXT" := FALSE; END_IF;
END_REGION

REGION Network 8: Extend Left Discharge Cylinder
   RUNG wire#powerrail
      Contact( "p45" )
      wire#w1
      S_Coil( "O_LDCEXT" )
   END_RUNG
   RUNG wire#powerrail
      Contact( "p59" )
   END_RUNG wire#w1
   // the same network as SCL:
   IF "p45" OR "p59" THEN "O_LDCEXT" := TRUE; END_IF;
END_REGION

REGION Network 9: Retract Center Discharge Cylinder
   RUNG wire#powerrail
      Contact( "p7" )
      wire#w1
      R_Coil( "O_CDCEXT" )
   END_RUNG
   RUNG wire#powerrail
      Contact( "p41" )
   END_RUNG wire#w1
   RUNG wire#powerrail
      Contact( "p68" )
   END_RUNG wire#w1
   // the same network as SCL:
   IF "p7" OR "p41" OR "p68" THEN "O_CDCEXT" := FALSE; END_IF;
END_REGION

REGION Network 10: Extend Center Discharge Cylinder
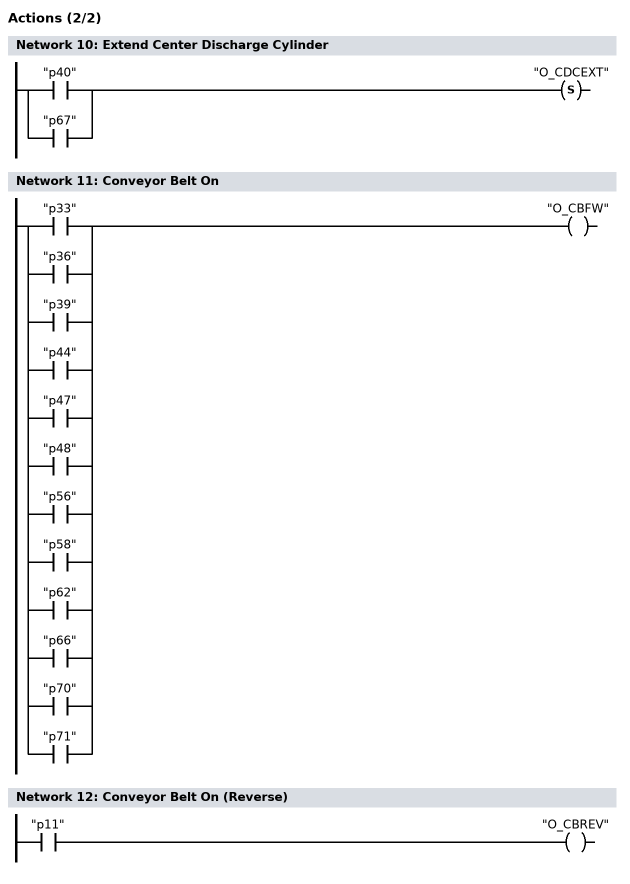
   RUNG wire#powerrail
      Contact( "p40" )
      wire#w1
      S_Coil( "O_CDCEXT" )
   END_RUNG
   RUNG wire#powerrail
      Contact( "p67" )
   END_RUNG wire#w1
   // the same network as SCL:
   IF "p40" OR "p67" THEN "O_CDCEXT" := TRUE; END_IF;
END_REGION

REGION Network 11: Conveyor Belt On
   RUNG wire#powerrail
      Contact( "p33" )
      wire#w1
      Coil( "O_CBFW" )
   END_RUNG
   RUNG wire#powerrail
      Contact( "p36" )
   END_RUNG wire#w1
   RUNG wire#powerrail
      Contact( "p39" )
   END_RUNG wire#w1
   RUNG wire#powerrail
      Contact( "p44" )
   END_RUNG wire#w1
   RUNG wire#powerrail
      Contact( "p47" )
   END_RUNG wire#w1
   RUNG wire#powerrail
      Contact( "p48" )
   END_RUNG wire#w1
   RUNG wire#powerrail
      Contact( "p56" )
   END_RUNG wire#w1
   RUNG wire#powerrail
      Contact( "p58" )
   END_RUNG wire#w1
   RUNG wire#powerrail
      Contact( "p62" )
   END_RUNG wire#w1
   RUNG wire#powerrail
      Contact( "p66" )
   END_RUNG wire#w1
   RUNG wire#powerrail
      Contact( "p70" )
   END_RUNG wire#w1
   RUNG wire#powerrail
      Contact( "p71" )
   END_RUNG wire#w1
   // the same network as SCL:
   "O_CBFW" := "p33" OR "p36" OR "p39" OR "p44" OR "p47" OR "p48" OR "p56" OR "p58" OR "p62" OR "p66" OR "p70" OR "p71";
END_REGION

REGION Network 12: Conveyor Belt On (Reverse)
   RUNG wire#powerrail
      Contact( "p11" )
      Coil( "O_CBREV" )
   END_RUNG
   // the same network as SCL:
   "O_CBREV" := "p11";
END_REGION
END_FUNCTION

// ===== PLC "Handling-Assembly-Storage"  CPU 1516-3 PN/DP =====

VAR_GLOBAL   // PLC tag table "IOTAGS"
   "I_SDO" AT %I1.0 : Bool;   // Safety Door Opened
   "I_SDC" AT %I1.1 : Bool;   // Safety Door Closed
   "I_AUHEXT" AT %I1.2 : Bool;   // Assembly Unit Holder Extended
   "I_AUHRET" AT %I1.3 : Bool;   // Assembly Unit Holder Retracted
   "I_INDARM" AT %I0.2 : Bool;   // Inductive Sensor Arm
   "I_ARMLOW" AT %I0.4 : Bool;   // Arm Lowered
   "I_ARMHIG" AT %I0.3 : Bool;   // Arm Raised
   "I_ARMRET" AT %I0.6 : Bool;   // Arm Retracted
   "I_ARMEXT" AT %I0.5 : Bool;   // Arm Extended
   "I_SUVE" AT %I2.0 : Bool;   // Storage Unit Vertical Encoder
   "I_SUILS" AT %I2.2 : Bool;   // Storage Unit Inferior Limit Switch
   "I_SUSLS" AT %I2.1 : Bool;   // Storage Unit Superior Limit Switch
   "I_SUEXT" AT %I2.3 : Bool;   // Storage Unit Extended
   "I_SURET" AT %I2.4 : Bool;   // Storage Unit Retracted
   "I_RELAY2" AT %I2.5 : Bool;   // Relay
   "I_SUHE" AT %I1.4 : Bool;   // Storage Unit Horizontal Encoder
   "I_SURLS" AT %I1.5 : Bool;   // Storage Unit Right Limit Switch
   "I_SULLS" AT %I1.6 : Bool;   // Storage Unit Left Limit Switch
   "I_SUARMALE" AT %I1.7 : Bool;   // Storage Unit Arm Alignment Encoder
   "O_SDO" AT %Q0.6 : Bool;   // Open Safety Door
   "O_SDC" AT %Q0.7 : Bool;   // Close Safety Door
   "O_AUHRET" AT %Q1.1 : Bool;   // Retract Assembly Unit Holder
   "O_AUHEXT" AT %Q1.0 : Bool;   // Extend Assembly Unit Holder
   "O_PRESSLOW" AT %Q1.2 : Bool;   // Lower Press
   "O_PRESSHIG" AT %Q1.3 : Bool;   // Raise Press
   "O_ARMHIG" AT %Q0.0 : Bool;   // Raise Arm
   "O_VACON" AT %Q0.1 : Bool;   // Turn Vacuum Gripper ON
   "O_ARMEXT" AT %Q0.2 : Bool;   // Extend Arm
   "O_ARMCCW" AT %Q0.3 : Bool;   // Turn Arm CCW
   "O_ARMCW" AT %Q0.4 : Bool;   // Turn Arm CW
   "O_SUEXT" AT %Q0.5 : Bool;   // Extend Storage Unit
   "O_SUUP" AT %Q1.6 : Bool;   // Move Storage Unit Upwards
   "O_SUDWN" AT %Q1.7 : Bool;   // Move Storage Unit Downwards
   "O_SURIGHT" AT %Q1.5 : Bool;   // Move Storage Unit to the Right
   "O_SULEFT" AT %Q1.4 : Bool;   // Move Storage Unit to the Left
END_VAR

VAR_GLOBAL   // PLC tag table "Places"
   "p14" AT %M0.0 : Bool;
   "p15" AT %M0.1 : Bool;
   "p16" AT %M0.2 : Bool;
   "p17" AT %M0.3 : Bool;
   "p18" AT %M0.4 : Bool;
   "p19" AT %M0.5 : Bool;
   "p20" AT %M0.6 : Bool;
   "p21" AT %M0.7 : Bool;
   "p22" AT %M1.0 : Bool;
   "p23" AT %M1.1 : Bool;
   "p24" AT %M1.2 : Bool;
   "p25" AT %M1.3 : Bool;
   "p26" AT %M1.4 : Bool;
   "p74" AT %M1.5 : Bool;
   "p75" AT %M1.6 : Bool;
   "p76" AT %M1.7 : Bool;
   "p77" AT %M2.0 : Bool;
   "p78" AT %M2.1 : Bool;
   "p79" AT %M2.2 : Bool;
   "p80" AT %M2.3 : Bool;
   "p81" AT %M2.4 : Bool;
   "p82" AT %M2.5 : Bool;
   "p83" AT %M2.6 : Bool;
   "p84" AT %M2.7 : Bool;
   "p85" AT %M3.0 : Bool;
   "p86" AT %M3.1 : Bool;
   "p87" AT %M3.2 : Bool;
   "p88" AT %M3.3 : Bool;
   "p89" AT %M3.4 : Bool;
   "p90" AT %M3.5 : Bool;
   "p91" AT %M3.6 : Bool;
   "p92" AT %M3.7 : Bool;
   "p93" AT %M4.0 : Bool;
   "p94" AT %M4.1 : Bool;
   "p95" AT %M4.2 : Bool;
   "p96" AT %M4.3 : Bool;
   "p97" AT %M4.4 : Bool;
   "p98" AT %M4.5 : Bool;
   "p99" AT %M4.6 : Bool;
   "p100" AT %M4.7 : Bool;
   "p101" AT %M5.0 : Bool;
   "p102" AT %M5.1 : Bool;
   "p103" AT %M5.2 : Bool;
   "p104" AT %M5.3 : Bool;
   "p105" AT %M5.4 : Bool;
   "p106" AT %M5.5 : Bool;
   "p107" AT %M5.6 : Bool;
   "p108" AT %M5.7 : Bool;
   "p109" AT %M6.0 : Bool;
   "p110" AT %M6.1 : Bool;
   "p111" AT %M6.2 : Bool;
   "p112" AT %M6.3 : Bool;
   "p113" AT %M6.4 : Bool;
   "p114" AT %M6.5 : Bool;
   "p115" AT %M6.6 : Bool;
   "p116" AT %M6.7 : Bool;
   "p117" AT %M7.0 : Bool;
   "p118" AT %M7.1 : Bool;
   "p119" AT %M7.2 : Bool;
   "p120" AT %M7.3 : Bool;
   "p121" AT %M7.4 : Bool;
   "p122" AT %M7.5 : Bool;
   "p123" AT %M7.6 : Bool;
   "p124" AT %M7.7 : Bool;
   "p125" AT %M8.0 : Bool;
   "p126" AT %M8.1 : Bool;
   "p127" AT %M8.2 : Bool;
   "p128" AT %M8.3 : Bool;
   "p129" AT %M8.4 : Bool;
   "p130" AT %M8.5 : Bool;
   "p131" AT %M8.6 : Bool;
   "p132" AT %M8.7 : Bool;
   "p133" AT %M9.0 : Bool;
   "p134" AT %M9.1 : Bool;
   "p135" AT %M9.2 : Bool;
   "p136" AT %M9.3 : Bool;
   "p137" AT %M9.4 : Bool;
   "p138" AT %M9.5 : Bool;
   "p139" AT %M9.6 : Bool;
   "p13" AT %M32.5 : Bool;
   "p140" AT %M35.6 : Bool;
   "p141" AT %M37.2 : Bool;
   "p145" AT %M37.3 : Bool;
   "p142" AT %M37.4 : Bool;
   "p143" AT %M37.5 : Bool;
   "p144" AT %M37.6 : Bool;
   "p146" AT %M37.7 : Bool;
END_VAR

VAR_GLOBAL   // PLC tag table "Transitions"
   "t8" AT %M10.5 : Bool;
   "t9" AT %M10.6 : Bool;
   "t10" AT %M10.7 : Bool;
   "t11" AT %M11.0 : Bool;
   "t12" AT %M11.1 : Bool;
   "t13" AT %M11.2 : Bool;
   "t14" AT %M11.3 : Bool;
   "t15" AT %M11.4 : Bool;
   "t16" AT %M11.5 : Bool;
   "t17" AT %M11.6 : Bool;
   "t72" AT %M11.7 : Bool;
   "t73" AT %M12.0 : Bool;
   "t74" AT %M12.1 : Bool;
   "t75" AT %M12.2 : Bool;
   "t76" AT %M12.3 : Bool;
   "t77" AT %M12.4 : Bool;
   "t78" AT %M12.5 : Bool;
   "t79" AT %M12.6 : Bool;
   "t80" AT %M12.7 : Bool;
   "t81" AT %M13.0 : Bool;
   "t82" AT %M13.1 : Bool;
   "t83" AT %M13.2 : Bool;
   "t84" AT %M13.3 : Bool;
   "t85" AT %M13.4 : Bool;
   "t86" AT %M13.5 : Bool;
   "t87" AT %M13.6 : Bool;
   "t88" AT %M13.7 : Bool;
   "t89" AT %M14.0 : Bool;
   "t90" AT %M14.1 : Bool;
   "t91" AT %M14.2 : Bool;
   "t92" AT %M14.3 : Bool;
   "t93" AT %M14.4 : Bool;
   "t94" AT %M14.5 : Bool;
   "t95" AT %M14.6 : Bool;
   "t96" AT %M14.7 : Bool;
   "t97" AT %M15.0 : Bool;
   "t98" AT %M15.1 : Bool;
   "t99" AT %M15.2 : Bool;
   "t100" AT %M15.3 : Bool;
   "t101" AT %M15.4 : Bool;
   "t102" AT %M15.5 : Bool;
   "t103" AT %M15.6 : Bool;
   "t104" AT %M15.7 : Bool;
   "t105" AT %M16.0 : Bool;
   "t106" AT %M16.1 : Bool;
   "t107" AT %M16.2 : Bool;
   "t108" AT %M16.3 : Bool;
   "t109" AT %M16.4 : Bool;
   "t110" AT %M16.5 : Bool;
   "t111" AT %M16.6 : Bool;
   "t112" AT %M16.7 : Bool;
   "t113" AT %M17.0 : Bool;
   "t114" AT %M17.1 : Bool;
   "t115" AT %M17.2 : Bool;
   "t116" AT %M17.3 : Bool;
   "t117" AT %M17.4 : Bool;
   "t118" AT %M17.5 : Bool;
   "t119" AT %M17.6 : Bool;
   "t120" AT %M17.7 : Bool;
   "t121" AT %M18.0 : Bool;
   "t122" AT %M18.1 : Bool;
   "t123" AT %M18.2 : Bool;
   "t124" AT %M18.3 : Bool;
   "t125" AT %M18.4 : Bool;
   "t126" AT %M18.5 : Bool;
   "t127" AT %M18.6 : Bool;
   "t128" AT %M18.7 : Bool;
   "t129" AT %M19.0 : Bool;
   "t130" AT %M19.1 : Bool;
   "t131" AT %M19.2 : Bool;
   "t132" AT %M19.3 : Bool;
   "t133" AT %M19.4 : Bool;
   "t134" AT %M19.5 : Bool;
   "t135" AT %M19.6 : Bool;
   "t136" AT %M19.7 : Bool;
   "t137" AT %M20.0 : Bool;
   "t138" AT %M20.1 : Bool;
   "t139" AT %M20.2 : Bool;
   "t140" AT %M20.3 : Bool;
   "t141" AT %M20.4 : Bool;
   "t142" AT %M20.5 : Bool;
   "t143" AT %M20.6 : Bool;
   "t144" AT %M20.7 : Bool;
   "t145" AT %M21.0 : Bool;
   "t146" AT %M21.1 : Bool;
   "t147" AT %M21.2 : Bool;
   "t148" AT %M21.3 : Bool;
   "t149" AT %M21.4 : Bool;
END_VAR

VAR_GLOBAL   // PLC tag table "Conditions"
   "b8" AT %M21.5 : Bool;
   "b9" AT %M21.6 : Bool;
   "b10" AT %M21.7 : Bool;
   "b11" AT %M22.0 : Bool;
   "b12" AT %M22.1 : Bool;
   "b13" AT %M22.2 : Bool;
   "b14" AT %M22.3 : Bool;
   "b15" AT %M22.4 : Bool;
   "b16" AT %M22.5 : Bool;
   "b17" AT %M22.6 : Bool;
   "b72" AT %M22.7 : Bool;
   "b73" AT %M23.0 : Bool;
   "b74" AT %M23.1 : Bool;
   "b75" AT %M23.2 : Bool;
   "b76" AT %M23.3 : Bool;
   "b77" AT %M23.4 : Bool;
   "b78" AT %M23.5 : Bool;
   "b79" AT %M23.6 : Bool;
   "b80" AT %M23.7 : Bool;
   "b81" AT %M24.0 : Bool;
   "b82" AT %M24.1 : Bool;
   "b83" AT %M24.2 : Bool;
   "b84" AT %M24.3 : Bool;
   "b85" AT %M24.4 : Bool;
   "b86" AT %M24.5 : Bool;
   "b87" AT %M24.6 : Bool;
   "b88" AT %M24.7 : Bool;
   "b89" AT %M25.0 : Bool;
   "b90" AT %M25.1 : Bool;
   "b91" AT %M25.2 : Bool;
   "b92" AT %M25.3 : Bool;
   "b93" AT %M25.4 : Bool;
   "b94" AT %M25.5 : Bool;
   "b95" AT %M25.6 : Bool;
   "b96" AT %M25.7 : Bool;
   "b97" AT %M26.0 : Bool;
   "b98" AT %M26.1 : Bool;
   "b99" AT %M26.2 : Bool;
   "b100" AT %M26.3 : Bool;
   "b101" AT %M26.4 : Bool;
   "b102" AT %M26.5 : Bool;
   "b103" AT %M26.6 : Bool;
   "b104" AT %M26.7 : Bool;
   "b105" AT %M27.0 : Bool;
   "b106" AT %M27.1 : Bool;
   "b107" AT %M27.2 : Bool;
   "b108" AT %M27.3 : Bool;
   "b109" AT %M27.4 : Bool;
   "b110" AT %M27.5 : Bool;
   "b111" AT %M27.6 : Bool;
   "b112" AT %M27.7 : Bool;
   "b113" AT %M28.0 : Bool;
   "b114" AT %M28.1 : Bool;
   "b115" AT %M28.2 : Bool;
   "b116" AT %M28.3 : Bool;
   "b117" AT %M28.4 : Bool;
   "b118" AT %M28.5 : Bool;
   "b119" AT %M28.6 : Bool;
   "b120" AT %M28.7 : Bool;
   "b121" AT %M29.0 : Bool;
   "b122" AT %M29.1 : Bool;
   "b123" AT %M29.2 : Bool;
   "b124" AT %M29.3 : Bool;
   "b125" AT %M29.4 : Bool;
   "b126" AT %M29.5 : Bool;
   "b127" AT %M29.6 : Bool;
   "b128" AT %M29.7 : Bool;
   "b129" AT %M30.0 : Bool;
   "b130" AT %M30.1 : Bool;
   "b131" AT %M30.2 : Bool;
   "b132" AT %M30.3 : Bool;
   "b133" AT %M30.4 : Bool;
   "b134" AT %M30.5 : Bool;
   "b135" AT %M30.6 : Bool;
   "b136" AT %M30.7 : Bool;
   "b137" AT %M31.0 : Bool;
   "b138" AT %M31.1 : Bool;
   "b139" AT %M31.2 : Bool;
   "b140" AT %M31.3 : Bool;
   "b141" AT %M31.4 : Bool;
   "b142" AT %M31.5 : Bool;
   "b143" AT %M31.6 : Bool;
   "b144" AT %M31.7 : Bool;
   "b145" AT %M32.0 : Bool;
   "b146" AT %M32.1 : Bool;
   "b147" AT %M32.2 : Bool;
   "b148" AT %M32.3 : Bool;
   "b149" AT %M32.4 : Bool;
   "b150" AT %M32.6 : Bool;
   "b151" AT %M32.7 : Bool;
   "b152" AT %M33.0 : Bool;
   "b153" AT %M33.1 : Bool;
   "b154" AT %M33.2 : Bool;
   "b0" AT %M10.2 : Bool;
   "b18" AT %M10.3 : Bool;
   "b45" AT %M33.4 : Bool;
   "b19" AT %M33.3 : Bool;
   "b71" AT %M33.5 : Bool;
   "b155" AT %M35.7 : Bool;
   "b156_StopAll" AT %M36.0 : Bool;
   "b157" AT %M36.1 : Bool;
   "b158" AT %M36.2 : Bool;
   "b159" AT %M36.3 : Bool;
   "b160" AT %M36.4 : Bool;
   "b161" AT %M36.5 : Bool;
   "b165" AT %M36.6 : Bool;
   "b164" AT %M36.7 : Bool;
   "b163" AT %M37.0 : Bool;
   "b162" AT %M37.1 : Bool;
END_VAR

VAR_GLOBAL   // PLC tag table "Auxiliar"
   "fromplc1_b0prev" AT %M9.7 : Bool;
   "frompl1_b18prev" AT %M10.0 : Bool;
   "frompl1_p18prev" AT %M10.1 : Bool;
   "frompl1_b19prev" AT %M10.4 : Bool;
   "b162aux" AT %M33.6 : Bool;
   "frompl1_b45prev" AT %M33.7 : Bool;
   "frompl1_b162prev" AT %M34.0 : Bool;
   "frompl1_b71prev" AT %M34.1 : Bool;
   "testecw" AT %M34.2 : Bool;
   "testeccw" AT %M34.3 : Bool;
   "tesete_extendarm" AT %M34.4 : Bool;
   "O_AUHEXTtest" AT %M34.5 : Bool;
   "O_AUHRETtest" AT %M34.6 : Bool;
   "O_PRESSHIGtest" AT %M34.7 : Bool;
   "O_PRESSLOWtest" AT %M35.0 : Bool;
   "I_SUHEprev" AT %M35.1 : Bool;
   "p118prev" AT %M35.2 : Bool;
   "p128prev" AT %M35.3 : Bool;
   "p115prev" AT %M35.4 : Bool;
   "p126prev" AT %M35.5 : Bool;
   "Stop" AT %M38.0 : Bool;
   "frompl1_btStopprev" AT %M38.1 : Bool;
END_VAR

VAR_GLOBAL CONSTANT   // PLC tag table "Auxiliar"
   "BELT_ANGLE_CW" : DInt := -1660;
   "PRESS_ANGLE" : DInt := -3320;
   "STORAGE_ANGLE" : DInt := -4935;
   "BELT_ANGLE_CCW" : DInt := -1720;
   "STORAGE_ANGLE_BEFORE" : DInt := -3800;
   "PRESS_ANGLE_BEFORE" : DInt := -3100;
   "PRESS_ANGLE_AFTER" : DInt := -3500;
END_VAR

// folder: Logging

DATA_BLOCK "IOVEC_TOPLC1"   // DB27
{ S7_Optimized_Access := 'FALSE' }
VERSION : 0.1
   VAR
      I_SDO : Bool;
      I_SDC : Bool;
      I_AUHEXT : Bool;
      I_AUHRET : Bool;
      I_INDARM : Bool;
      I_ARMLOW : Bool;
      I_ARMHIG : Bool;
      I_ARMRET : Bool;
      I_ARMEXT : Bool;
      I_SUVE : Bool;
      I_SUILS : Bool;
      I_SUSLS : Bool;
      I_SUEXT : Bool;
      I_SURET : Bool;
      I_RELAY2 : Bool;
      I_SUHE : Bool;
      I_SURLS : Bool;
      I_SULLS : Bool;
      I_SUARMALE : Bool;
      O_SDO : Bool;
      O_SDC : Bool;
      O_AUHRET : Bool;
      O_AUHEXT : Bool;
      O_PRESSLOW : Bool;
      O_PRESSHIG : Bool;
      O_ARMHIG : Bool;
      O_VACON : Bool;
      O_ARMEXT : Bool;
      O_ARMCCW : Bool;
      O_ARMCW : Bool;
      O_SUEXT : Bool;
      O_SUUP : Bool;
      O_SUDWN : Bool;
      O_SURIGHT : Bool;
      O_SULEFT : Bool;
   END_VAR
BEGIN
END_DATA_BLOCK

// folder: PetriNet

DATA_BLOCK "FROM_PLC1"   // DB4
{ S7_Optimized_Access := 'FALSE' }
VERSION : 0.1
   VAR
      b0 : Bool;
      b18 : Bool;
      b19 : Bool;
      b71 : Bool;
      b45 : Bool;
      b162 : Bool;
      btStopOn : Bool;
      btStopOff : Bool;
   END_VAR
BEGIN
END_DATA_BLOCK

DATA_BLOCK "TO_PLC1"   // DB5
{ S7_Optimized_Access := 'FALSE' }
VERSION : 0.1
   VAR
      p13 : Bool;
      p17 : Bool;
      p26 : Bool;
      p14 : Bool;
      p18 : Bool;
      p107 : Bool;
      p0 : Bool;
      b162aux : Bool;
   END_VAR
BEGIN
END_DATA_BLOCK

// folder: PetriNet/TimedTransitions

DATA_BLOCK "t8_time"   // DB1
{ S7_Optimized_Access := 'TRUE' }
AUTHOR : Simatic
FAMILY : IEC
NAME : IEC_TMR
VERSION : 1.0
// stored: InstanceOfName IEC_TIMER
"IEC_TIMER"
BEGIN
END_DATA_BLOCK

DATA_BLOCK "t14_time"   // DB2
{ S7_Optimized_Access := 'TRUE' }
AUTHOR : Simatic
FAMILY : IEC
NAME : IEC_TMR
VERSION : 1.0
// stored: InstanceOfName IEC_TIMER
"IEC_TIMER"
BEGIN
END_DATA_BLOCK

DATA_BLOCK "t16_time"   // DB3
{ S7_Optimized_Access := 'TRUE' }
AUTHOR : Simatic
FAMILY : IEC
NAME : IEC_TMR
VERSION : 1.0
// stored: InstanceOfName IEC_TIMER
"IEC_TIMER"
BEGIN
END_DATA_BLOCK

DATA_BLOCK "t73_time"   // DB6
{ S7_Optimized_Access := 'TRUE' }
AUTHOR : Simatic
FAMILY : IEC
NAME : IEC_TMR
VERSION : 1.0
// stored: InstanceOfName IEC_TIMER
"IEC_TIMER"
BEGIN
END_DATA_BLOCK

DATA_BLOCK "t74_time"   // DB7
{ S7_Optimized_Access := 'TRUE' }
AUTHOR : Simatic
FAMILY : IEC
NAME : IEC_TMR
VERSION : 1.0
// stored: InstanceOfName IEC_TIMER
"IEC_TIMER"
BEGIN
END_DATA_BLOCK

DATA_BLOCK "t75_time"   // DB8
{ S7_Optimized_Access := 'TRUE' }
AUTHOR : Simatic
FAMILY : IEC
NAME : IEC_TMR
VERSION : 1.0
// stored: InstanceOfName IEC_TIMER
"IEC_TIMER"
BEGIN
END_DATA_BLOCK

DATA_BLOCK "t76_time"   // DB9
{ S7_Optimized_Access := 'TRUE' }
AUTHOR : Simatic
FAMILY : IEC
NAME : IEC_TMR
VERSION : 1.0
// stored: InstanceOfName IEC_TIMER
"IEC_TIMER"
BEGIN
END_DATA_BLOCK

DATA_BLOCK "t78_time"   // DB10
{ S7_Optimized_Access := 'TRUE' }
AUTHOR : Simatic
FAMILY : IEC
NAME : IEC_TMR
VERSION : 1.0
// stored: InstanceOfName IEC_TIMER
"IEC_TIMER"
BEGIN
END_DATA_BLOCK

DATA_BLOCK "t79_time"   // DB11
{ S7_Optimized_Access := 'TRUE' }
AUTHOR : Simatic
FAMILY : IEC
NAME : IEC_TMR
VERSION : 1.0
// stored: InstanceOfName IEC_TIMER
"IEC_TIMER"
BEGIN
END_DATA_BLOCK

DATA_BLOCK "t80_time"   // DB12
{ S7_Optimized_Access := 'TRUE' }
AUTHOR : Simatic
FAMILY : IEC
NAME : IEC_TMR
VERSION : 1.0
// stored: InstanceOfName IEC_TIMER
"IEC_TIMER"
BEGIN
END_DATA_BLOCK

DATA_BLOCK "t81_time"   // DB13
{ S7_Optimized_Access := 'TRUE' }
AUTHOR : Simatic
FAMILY : IEC
NAME : IEC_TMR
VERSION : 1.0
// stored: InstanceOfName IEC_TIMER
"IEC_TIMER"
BEGIN
END_DATA_BLOCK

DATA_BLOCK "t83_time"   // DB15
{ S7_Optimized_Access := 'TRUE' }
AUTHOR : Simatic
FAMILY : IEC
NAME : IEC_TMR
VERSION : 1.0
// stored: InstanceOfName IEC_TIMER
"IEC_TIMER"
BEGIN
END_DATA_BLOCK

DATA_BLOCK "t86_time"   // DB16
{ S7_Optimized_Access := 'TRUE' }
AUTHOR : Simatic
FAMILY : IEC
NAME : IEC_TMR
VERSION : 1.0
// stored: InstanceOfName IEC_TIMER
"IEC_TIMER"
BEGIN
END_DATA_BLOCK

DATA_BLOCK "t87_time"   // DB17
{ S7_Optimized_Access := 'TRUE' }
AUTHOR : Simatic
FAMILY : IEC
NAME : IEC_TMR
VERSION : 1.0
// stored: InstanceOfName IEC_TIMER
"IEC_TIMER"
BEGIN
END_DATA_BLOCK

DATA_BLOCK "t88_time"   // DB18
{ S7_Optimized_Access := 'TRUE' }
AUTHOR : Simatic
FAMILY : IEC
NAME : IEC_TMR
VERSION : 1.0
// stored: InstanceOfName IEC_TIMER
"IEC_TIMER"
BEGIN
END_DATA_BLOCK

DATA_BLOCK "t89_time"   // DB19
{ S7_Optimized_Access := 'TRUE' }
AUTHOR : Simatic
FAMILY : IEC
NAME : IEC_TMR
VERSION : 1.0
// stored: InstanceOfName IEC_TIMER
"IEC_TIMER"
BEGIN
END_DATA_BLOCK

DATA_BLOCK "t90_time"   // DB20
{ S7_Optimized_Access := 'TRUE' }
AUTHOR : Simatic
FAMILY : IEC
NAME : IEC_TMR
VERSION : 1.0
// stored: InstanceOfName IEC_TIMER
"IEC_TIMER"
BEGIN
END_DATA_BLOCK

DATA_BLOCK "t91_time"   // DB21
{ S7_Optimized_Access := 'TRUE' }
AUTHOR : Simatic
FAMILY : IEC
NAME : IEC_TMR
VERSION : 1.0
// stored: InstanceOfName IEC_TIMER
"IEC_TIMER"
BEGIN
END_DATA_BLOCK

DATA_BLOCK "t94_time"   // DB22
{ S7_Optimized_Access := 'TRUE' }
AUTHOR : Simatic
FAMILY : IEC
NAME : IEC_TMR
VERSION : 1.0
// stored: InstanceOfName IEC_TIMER
"IEC_TIMER"
BEGIN
END_DATA_BLOCK

DATA_BLOCK "t98_time"   // DB23
{ S7_Optimized_Access := 'TRUE' }
AUTHOR : Simatic
FAMILY : IEC
NAME : IEC_TMR
VERSION : 1.0
// stored: InstanceOfName IEC_TIMER
"IEC_TIMER"
BEGIN
END_DATA_BLOCK

DATA_BLOCK "t99_time"   // DB24
{ S7_Optimized_Access := 'TRUE' }
AUTHOR : Simatic
FAMILY : IEC
NAME : IEC_TMR
VERSION : 1.0
// stored: InstanceOfName IEC_TIMER
"IEC_TIMER"
BEGIN
END_DATA_BLOCK

DATA_BLOCK "t103_time"   // DB25
{ S7_Optimized_Access := 'TRUE' }
AUTHOR : Simatic
FAMILY : IEC
NAME : IEC_TMR
VERSION : 1.0
// stored: InstanceOfName IEC_TIMER
"IEC_TIMER"
BEGIN
END_DATA_BLOCK

DATA_BLOCK "t105_time"   // DB26
{ S7_Optimized_Access := 'TRUE' }
AUTHOR : Simatic
FAMILY : IEC
NAME : IEC_TMR
VERSION : 1.0
// stored: InstanceOfName IEC_TIMER
"IEC_TIMER"
BEGIN
END_DATA_BLOCK

DATA_BLOCK "t140_time"   // DB33
{ S7_Optimized_Access := 'TRUE' }
AUTHOR : Simatic
FAMILY : IEC
NAME : IEC_TMR
VERSION : 1.0
// stored: InstanceOfName IEC_TIMER
"IEC_TIMER"
BEGIN
END_DATA_BLOCK

DATA_BLOCK "t141_time"   // DB34
{ S7_Optimized_Access := 'TRUE' }
AUTHOR : Simatic
FAMILY : IEC
NAME : IEC_TMR
VERSION : 1.0
// stored: InstanceOfName IEC_TIMER
"IEC_TIMER"
BEGIN
END_DATA_BLOCK

DATA_BLOCK "t142_time"   // DB35
{ S7_Optimized_Access := 'TRUE' }
AUTHOR : Simatic
FAMILY : IEC
NAME : IEC_TMR
VERSION : 1.0
// stored: InstanceOfName IEC_TIMER
"IEC_TIMER"
BEGIN
END_DATA_BLOCK

DATA_BLOCK "t143_time"   // DB36
{ S7_Optimized_Access := 'TRUE' }
AUTHOR : Simatic
FAMILY : IEC
NAME : IEC_TMR
VERSION : 1.0
// stored: InstanceOfName IEC_TIMER
"IEC_TIMER"
BEGIN
END_DATA_BLOCK

DATA_BLOCK "t144_time"   // DB37
{ S7_Optimized_Access := 'TRUE' }
AUTHOR : Simatic
FAMILY : IEC
NAME : IEC_TMR
VERSION : 1.0
// stored: InstanceOfName IEC_TIMER
"IEC_TIMER"
BEGIN
END_DATA_BLOCK

// folder: System blocks/Program resources

DATA_BLOCK "HalfPieceCounter"   // DB14
{ S7_Optimized_Access := 'TRUE' }
AUTHOR : Simatic
FAMILY : IEC
NAME : CNTR
VERSION : 1.0
// stored: InstanceOfName IEC_COUNTER
"IEC_COUNTER"
BEGIN
END_DATA_BLOCK

DATA_BLOCK "COUNTER1"   // DB28
{ S7_Optimized_Access := 'TRUE' }
AUTHOR : Simatic
FAMILY : IEC
NAME : CNTR
VERSION : 1.0
// stored: InstanceOfName IEC_COUNTER
"IEC_COUNTER"
BEGIN
END_DATA_BLOCK

DATA_BLOCK "COUNTER2"   // DB29
{ S7_Optimized_Access := 'TRUE' }
AUTHOR : Simatic
FAMILY : IEC
NAME : CNTR
VERSION : 1.0
// stored: InstanceOfName IEC_COUNTER
"IEC_COUNTER"
BEGIN
END_DATA_BLOCK

DATA_BLOCK "COUNTER3"   // DB30
{ S7_Optimized_Access := 'TRUE' }
AUTHOR : Simatic
FAMILY : IEC
NAME : CNTR
VERSION : 1.0
// stored: InstanceOfName IEC_COUNTER
"IEC_COUNTER"
BEGIN
END_DATA_BLOCK

DATA_BLOCK "COUNTER4"   // DB31
{ S7_Optimized_Access := 'TRUE' }
AUTHOR : Simatic
FAMILY : IEC
NAME : CNTR
VERSION : 1.0
// stored: InstanceOfName IEC_COUNTER
"IEC_COUNTER"
BEGIN
END_DATA_BLOCK

DATA_BLOCK "COUNTER5"   // DB32
{ S7_Optimized_Access := 'TRUE' }
AUTHOR : Simatic
FAMILY : IEC
NAME : CNTR
VERSION : 1.0
// stored: InstanceOfName IEC_COUNTER
"IEC_COUNTER"
BEGIN
END_DATA_BLOCK

// folder: (top level)

ORGANIZATION_BLOCK "Main"   // OB1, LAD, ProgramCycle
TITLE = "Main Program Sweep (Cycle)"
{ S7_Optimized_Access := 'TRUE' }
VERSION : 0.1
   VAR_INPUT
      Initial_Call : Bool;   // Initial call of this OB
      Remanence : Bool;   // =True, if remanent data are available
   END_VAR
   VAR_TEMP   // added for the SCL form of the ladder/FBD networks
      _w1 : Bool;
      _w2 : Bool;
      _w3 : Bool;
      _w4 : Bool;
      _w5 : Bool;
      _w6 : Bool;
      _w7 : Bool;
   END_VAR
BEGIN

REGION Network 1
   // get from plc 1
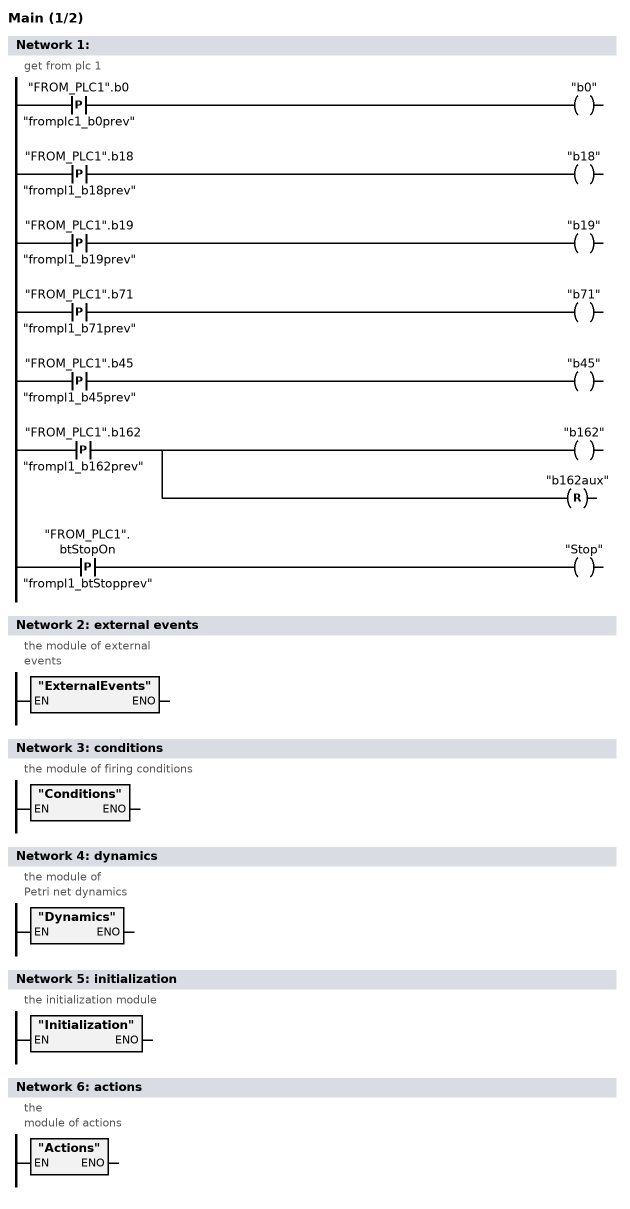
   RUNG wire#powerrail
      P_Contact(operand := "FROM_PLC1".b0, bit := "fromplc1_b0prev")
      Coil( "b0" )
   END_RUNG
   RUNG wire#powerrail
      P_Contact(operand := "FROM_PLC1".b18, bit := "frompl1_b18prev")
      Coil( "b18" )
   END_RUNG
   RUNG wire#powerrail
      P_Contact(operand := "FROM_PLC1".b19, bit := "frompl1_b19prev")
      Coil( "b19" )
   END_RUNG
   RUNG wire#powerrail
      P_Contact(operand := "FROM_PLC1".b71, bit := "frompl1_b71prev")
      Coil( "b71" )
   END_RUNG
   RUNG wire#powerrail
      P_Contact(operand := "FROM_PLC1".b45, bit := "frompl1_b45prev")
      Coil( "b45" )
   END_RUNG
   RUNG wire#powerrail
      P_Contact(operand := "FROM_PLC1".b162, bit := "frompl1_b162prev")
      wire#w1
      Coil( "b162" )
   END_RUNG
   RUNG wire#w1
      R_Coil( "b162aux" )
   END_RUNG
   RUNG wire#powerrail
      P_Contact(operand := "FROM_PLC1".btStopOn, bit := "frompl1_btStopprev")
      Coil( "Stop" )
   END_RUNG
   // the same network as SCL:
   #_w1 := "FROM_PLC1".b0 AND NOT "fromplc1_b0prev";   // rising edge of "FROM_PLC1".b0
   "fromplc1_b0prev" := "FROM_PLC1".b0;
   "b0" := #_w1;
   #_w2 := "FROM_PLC1".b18 AND NOT "frompl1_b18prev";   // rising edge of "FROM_PLC1".b18
   "frompl1_b18prev" := "FROM_PLC1".b18;
   "b18" := #_w2;
   #_w3 := "FROM_PLC1".b19 AND NOT "frompl1_b19prev";   // rising edge of "FROM_PLC1".b19
   "frompl1_b19prev" := "FROM_PLC1".b19;
   "b19" := #_w3;
   #_w4 := "FROM_PLC1".b71 AND NOT "frompl1_b71prev";   // rising edge of "FROM_PLC1".b71
   "frompl1_b71prev" := "FROM_PLC1".b71;
   "b71" := #_w4;
   #_w5 := "FROM_PLC1".b45 AND NOT "frompl1_b45prev";   // rising edge of "FROM_PLC1".b45
   "frompl1_b45prev" := "FROM_PLC1".b45;
   "b45" := #_w5;
   #_w6 := "FROM_PLC1".b162 AND NOT "frompl1_b162prev";   // rising edge of "FROM_PLC1".b162
   "frompl1_b162prev" := "FROM_PLC1".b162;
   "b162" := #_w6;
   IF #_w6 THEN "b162aux" := FALSE; END_IF;
   #_w7 := "FROM_PLC1".btStopOn AND NOT "frompl1_btStopprev";   // rising edge of "FROM_PLC1".btStopOn
   "frompl1_btStopprev" := "FROM_PLC1".btStopOn;
   "Stop" := #_w7;
END_REGION

REGION Network 2: external events
   // the module of external
   // events
   RUNG wire#powerrail
      "ExternalEvents"()
   END_RUNG
   // the same network as SCL:
   "ExternalEvents"();
END_REGION

REGION Network 3: conditions
   // the module of firing conditions
   RUNG wire#powerrail
      "Conditions"()
   END_RUNG
   // the same network as SCL:
   "Conditions"();
END_REGION

REGION Network 4: dynamics
   // the module of
   // Petri net dynamics
   RUNG wire#powerrail
      "Dynamics"()
   END_RUNG
   // the same network as SCL:
   "Dynamics"();
END_REGION

REGION Network 5: initialization
   // the initialization module
   RUNG wire#powerrail
      "Initialization"()
   END_RUNG
   // the same network as SCL:
   "Initialization"();
END_REGION

REGION Network 6: actions
   // the
   // module of actions
   RUNG wire#powerrail
      "Actions"()
   END_RUNG
   // the same network as SCL:
   "Actions"();
END_REGION

REGION Network 7
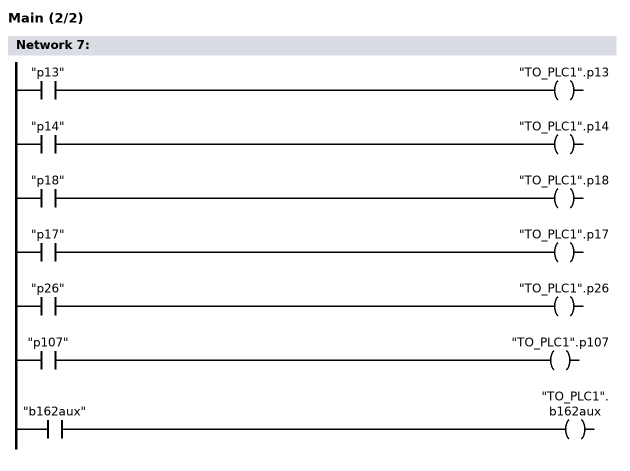
   RUNG wire#powerrail
      Contact( "p13" )
      Coil( "TO_PLC1".p13 )
   END_RUNG
   RUNG wire#powerrail
      Contact( "p14" )
      Coil( "TO_PLC1".p14 )
   END_RUNG
   RUNG wire#powerrail
      Contact( "p18" )
      Coil( "TO_PLC1".p18 )
   END_RUNG
   RUNG wire#powerrail
      Contact( "p17" )
      Coil( "TO_PLC1".p17 )
   END_RUNG
   RUNG wire#powerrail
      Contact( "p26" )
      Coil( "TO_PLC1".p26 )
   END_RUNG
   RUNG wire#powerrail
      Contact( "p107" )
      Coil( "TO_PLC1".p107 )
   END_RUNG
   RUNG wire#powerrail
      Contact( "b162aux" )
      Coil( "TO_PLC1".b162aux )
   END_RUNG
   // the same network as SCL:
   "TO_PLC1".p13 := "p13";
   "TO_PLC1".p14 := "p14";
   "TO_PLC1".p18 := "p18";
   "TO_PLC1".p17 := "p17";
   "TO_PLC1".p26 := "p26";
   "TO_PLC1".p107 := "p107";
   "TO_PLC1".b162aux := "b162aux";
END_REGION

REGION Network 8 (SCL): Set IOVECs TO PLC1
   "IOVEC_TOPLC1".I_SDO := "I_SDO";
   "IOVEC_TOPLC1".I_SDC := "I_SDC";
   "IOVEC_TOPLC1".I_AUHEXT := "I_AUHEXT";
   "IOVEC_TOPLC1".I_AUHRET := "I_AUHRET";
   "IOVEC_TOPLC1".I_INDARM := "I_INDARM";
   "IOVEC_TOPLC1".I_ARMLOW := "I_ARMLOW";
   "IOVEC_TOPLC1".I_ARMHIG := "I_ARMHIG";
   "IOVEC_TOPLC1".I_ARMRET := "I_ARMRET";
   "IOVEC_TOPLC1".I_ARMEXT := "I_ARMEXT";
   "IOVEC_TOPLC1".I_SUVE := "I_SUVE";
   "IOVEC_TOPLC1".I_SUILS := "I_SUILS";
   "IOVEC_TOPLC1".I_SUSLS := "I_SUSLS";
   "IOVEC_TOPLC1".I_SUEXT := "I_SUEXT";
   "IOVEC_TOPLC1".I_SURET := "I_SURET";
   "IOVEC_TOPLC1".I_RELAY2 := "I_RELAY2";
   "IOVEC_TOPLC1".I_SUHE := "I_SUHE";
   "IOVEC_TOPLC1".I_SURLS := "I_SURLS";
   "IOVEC_TOPLC1".I_SULLS := "I_SULLS";
   "IOVEC_TOPLC1".I_SUARMALE := "I_SUARMALE";
   "IOVEC_TOPLC1".O_SDO := "O_SDO";
   "IOVEC_TOPLC1".O_SDC := "O_SDC";
   "IOVEC_TOPLC1".O_AUHRET := "O_AUHRET";
   "IOVEC_TOPLC1".O_AUHEXT := "O_AUHEXT";
   "IOVEC_TOPLC1".O_PRESSLOW := "O_PRESSLOW";
   "IOVEC_TOPLC1".O_PRESSHIG := "O_PRESSHIG";
   "IOVEC_TOPLC1".O_ARMHIG := "O_ARMHIG";
   "IOVEC_TOPLC1".O_VACON := "O_VACON";
   "IOVEC_TOPLC1".O_ARMEXT := "O_ARMEXT";
   "IOVEC_TOPLC1".O_ARMCCW := "O_ARMCCW";
   "IOVEC_TOPLC1".O_ARMCW := "O_ARMCW";
   "IOVEC_TOPLC1".O_SUEXT := "O_SUEXT";
   "IOVEC_TOPLC1".O_SUUP := "O_SUUP";
   "IOVEC_TOPLC1".O_SUDWN := "O_SUDWN";
   "IOVEC_TOPLC1".O_SURIGHT := "O_SURIGHT";
   "IOVEC_TOPLC1".O_SULEFT := "O_SULEFT";
END_REGION
END_ORGANIZATION_BLOCK

// folder: PetriNet

FUNCTION "ExternalEvents" : Void   // FC1, LAD
{ S7_Optimized_Access := 'TRUE' }
VERSION : 0.1
BEGIN
END_FUNCTION

FUNCTION "Conditions" : Void   // FC2, LAD
{ S7_Optimized_Access := 'TRUE' }
VERSION : 0.1
BEGIN

REGION Network 1: initialization
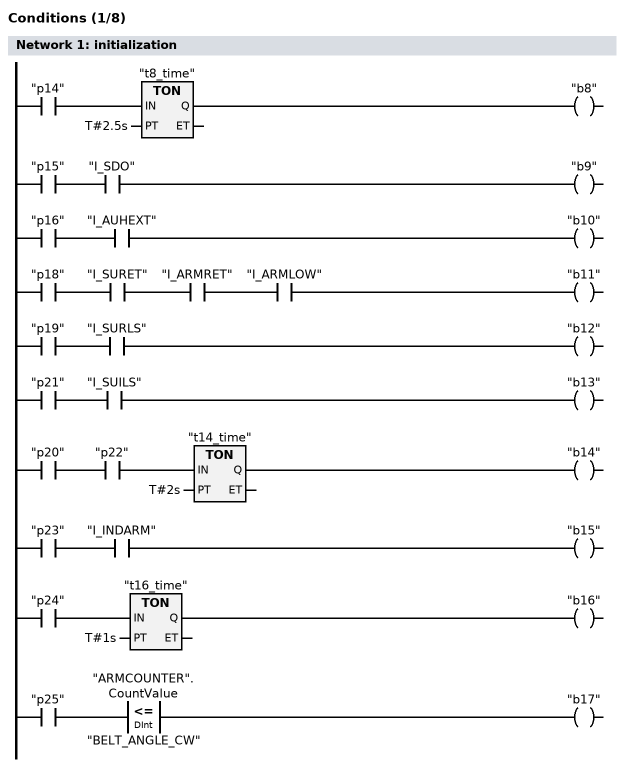
   "t8_time".TON(IN := "p14", PT := T#2.5s);
   "b8" := "t8_time".Q;
   "b9" := "p15" AND "I_SDO";
   "b10" := "p16" AND "I_AUHEXT";
   "b11" := "p18" AND "I_SURET" AND "I_ARMRET" AND "I_ARMLOW";
   "b12" := "p19" AND "I_SURLS";
   "b13" := "p21" AND "I_SUILS";
   "t14_time".TON(IN := "p20" AND "p22", PT := T#2s);
   "b14" := "t14_time".Q;
   "b15" := "p23" AND "I_INDARM";
   "t16_time".TON(IN := "p24", PT := T#1s);
   "b16" := "t16_time".Q;
   "b17" := "p25" AND ("ARMCOUNTER".CountValue <= "BELT_ANGLE_CW");
END_REGION

REGION Network 2: Arm Belt to Press
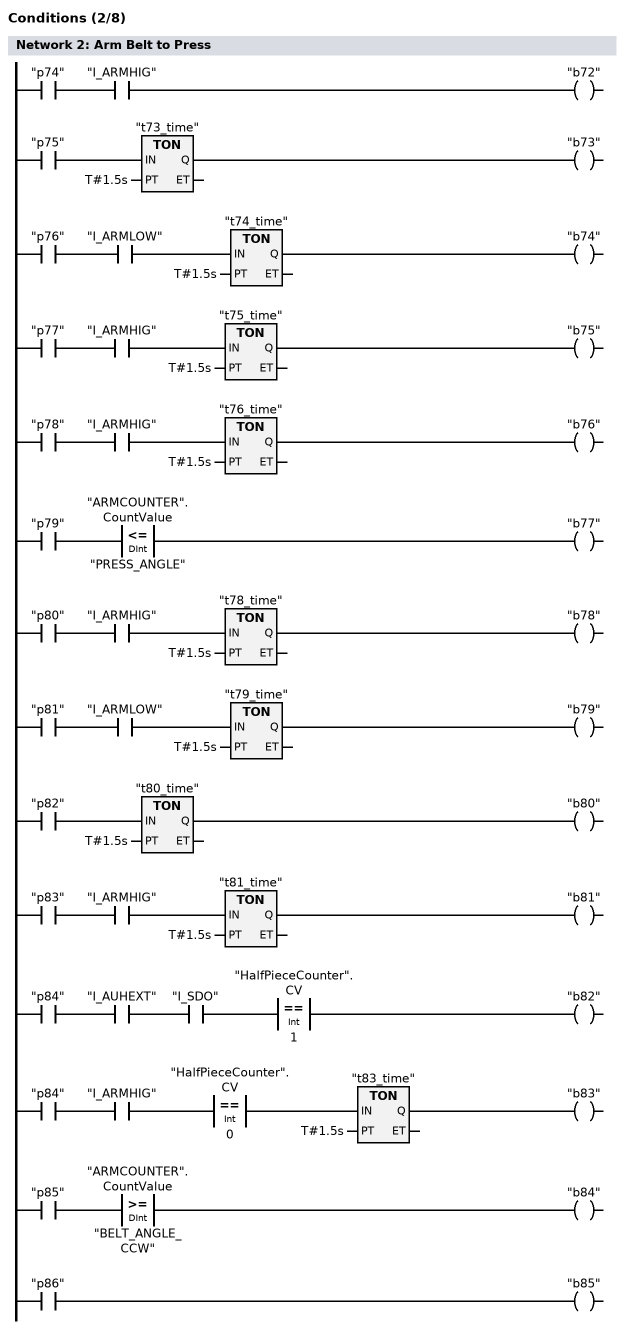
   "b72" := "p74" AND "I_ARMHIG";
   "t73_time".TON(IN := "p75", PT := T#1.5s);
   "b73" := "t73_time".Q;
   "t74_time".TON(IN := "p76" AND "I_ARMLOW", PT := T#1.5s);
   "b74" := "t74_time".Q;
   "t75_time".TON(IN := "p77" AND "I_ARMHIG", PT := T#1.5s);
   "b75" := "t75_time".Q;
   "t76_time".TON(IN := "p78" AND "I_ARMHIG", PT := T#1.5s);
   "b76" := "t76_time".Q;
   "b77" := "p79" AND ("ARMCOUNTER".CountValue <= "PRESS_ANGLE");
   "t78_time".TON(IN := "p80" AND "I_ARMHIG", PT := T#1.5s);
   "b78" := "t78_time".Q;
   "t79_time".TON(IN := "p81" AND "I_ARMLOW", PT := T#1.5s);
   "b79" := "t79_time".Q;
   "t80_time".TON(IN := "p82", PT := T#1.5s);
   "b80" := "t80_time".Q;
   "t81_time".TON(IN := "p83" AND "I_ARMHIG", PT := T#1.5s);
   "b81" := "t81_time".Q;
   "b82" := "p84" AND "I_AUHEXT" AND "I_SDO" AND ("HalfPieceCounter".CV = 1);
   "t83_time".TON(IN := "p84" AND "I_ARMHIG" AND ("HalfPieceCounter".CV = 0), PT := T#1.5s);
   "b83" := "t83_time".Q;
   "b84" := "p85" AND ("ARMCOUNTER".CountValue >= "BELT_ANGLE_CCW");
   "b85" := "p86";
END_REGION

REGION Network 3: Assembly Unit
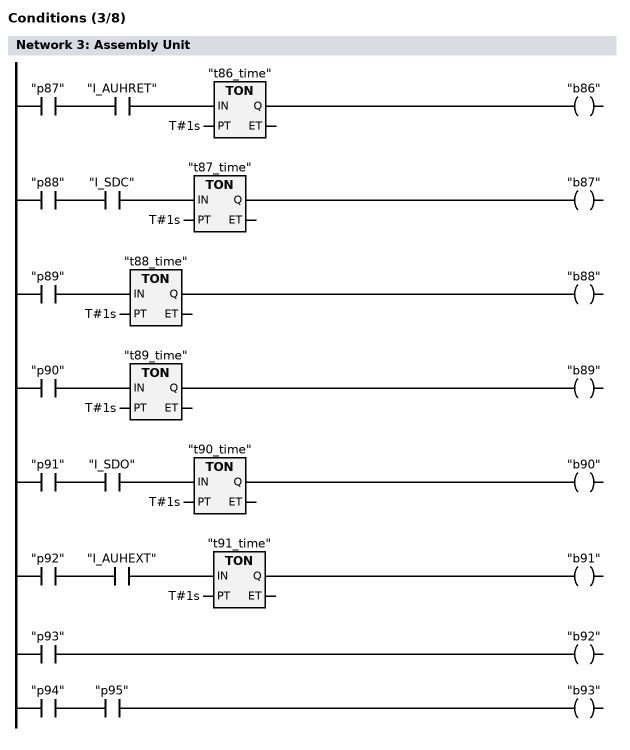
   "t86_time".TON(IN := "p87" AND "I_AUHRET", PT := T#1s);
   "b86" := "t86_time".Q;
   "t87_time".TON(IN := "p88" AND "I_SDC", PT := T#1s);
   "b87" := "t87_time".Q;
   "t88_time".TON(IN := "p89", PT := T#1s);
   "b88" := "t88_time".Q;
   "t89_time".TON(IN := "p90", PT := T#1s);
   "b89" := "t89_time".Q;
   "t90_time".TON(IN := "p91" AND "I_SDO", PT := T#1s);
   "b90" := "t90_time".Q;
   "t91_time".TON(IN := "p92" AND "I_AUHEXT", PT := T#1s);
   "b91" := "t91_time".Q;
   "b92" := "p93";
   "b93" := "p94" AND "p95";
END_REGION

REGION Network 4: Arm Press to Storage Unit
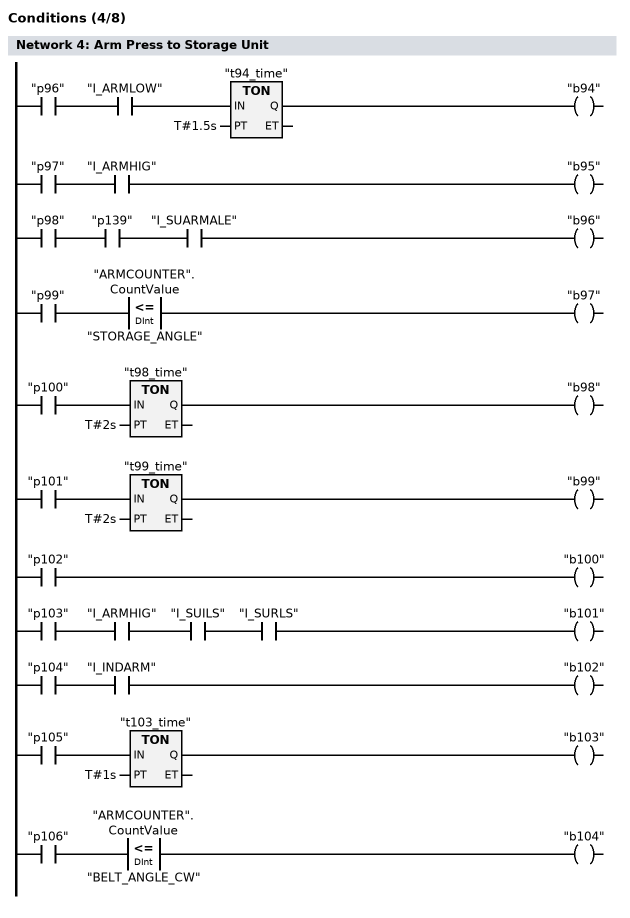
   "t94_time".TON(IN := "p96" AND "I_ARMLOW", PT := T#1.5s);
   "b94" := "t94_time".Q;
   "b95" := "p97" AND "I_ARMHIG";
   "b96" := "p98" AND "p139" AND "I_SUARMALE";
   "b97" := "p99" AND ("ARMCOUNTER".CountValue <= "STORAGE_ANGLE");
   "t98_time".TON(IN := "p100", PT := T#2s);
   "b98" := "t98_time".Q;
   "t99_time".TON(IN := "p101", PT := T#2s);
   "b99" := "t99_time".Q;
   "b100" := "p102";
   "b101" := "p103" AND "I_ARMHIG" AND "I_SUILS" AND "I_SURLS";
   "b102" := "p104" AND "I_INDARM";
   "t103_time".TON(IN := "p105", PT := T#1s);
   "b103" := "t103_time".Q;
   "b104" := "p106" AND ("ARMCOUNTER".CountValue <= "BELT_ANGLE_CW");
END_REGION

REGION Network 5: Storage Y
